// TIA Portal V17 export
// export: Created 2022-03-12T16:05:27.8169496Z, ExportSetting WithDefaults, DisplayName Totally Integrated Automation Portal, DisplayVersion V17, DisplayName TIA Portal Openness, DisplayVersion V17, DisplayName TIA Portal Version Control Interface, DisplayVersion V17, DisplayName STEP 7 Professional, DisplayVersion V17, DisplayName STEP 7 Safety, DisplayVersion V17, DisplayName WinCC Advanced / Unified PC, DisplayVersion V17
FUNCTION_BLOCK "EM01_02_PackML_ModuleSum"   // FB31662, LAD
TITLE = EM01_02_PackML_ModuleSum
{ S7_Optimized_Access := 'TRUE' }
AUTHOR : tech.team.motioncontrol@siemens.com
FAMILY : CPG
VERSION : 1.1
// Support: tech.team.motioncontrol@siemens.com
// stored: AutoNumber true, IsIECCheckEnabled false, IsRetainMemResEnabled false, MemoryReserve 100, SetENOAutomatically false, UDAEnableTagReadback false
   VAR
      statDummyBool { ExternalAccessible := 'False'; ExternalVisible := 'False'; ExternalWritable := 'False'} : Bool;   // dummy bool - placeholder
   END_VAR
BEGIN

REGION Network 1: EM - Reset Command
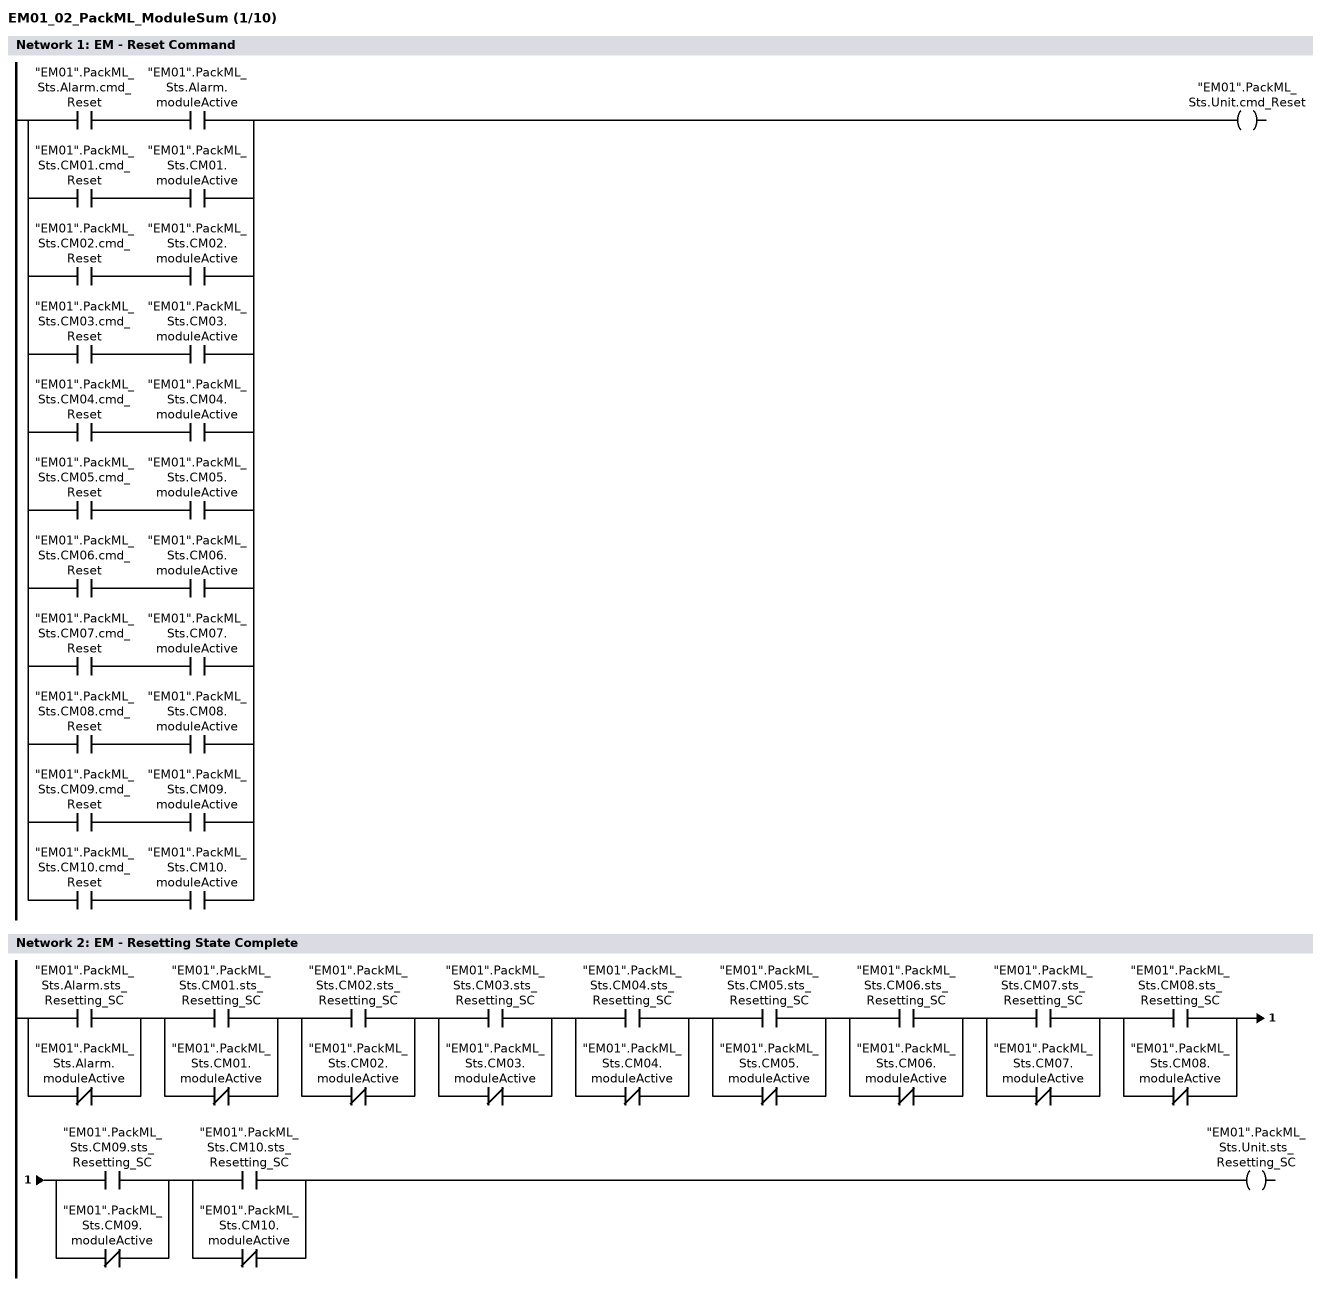
   RUNG wire#powerrail
      Contact( "EM01".PackML_Sts.Alarm.cmd_Reset )
      Contact( "EM01".PackML_Sts.Alarm.moduleActive )
      wire#w1
      Coil( "EM01".PackML_Sts.Unit.cmd_Reset )
   END_RUNG
   RUNG wire#powerrail
      Contact( "EM01".PackML_Sts.CM01.cmd_Reset )
      Contact( "EM01".PackML_Sts.CM01.moduleActive )
   END_RUNG wire#w1
   RUNG wire#powerrail
      Contact( "EM01".PackML_Sts.CM02.cmd_Reset )
      Contact( "EM01".PackML_Sts.CM02.moduleActive )
   END_RUNG wire#w1
   RUNG wire#powerrail
      Contact( "EM01".PackML_Sts.CM03.cmd_Reset )
      Contact( "EM01".PackML_Sts.CM03.moduleActive )
   END_RUNG wire#w1
   RUNG wire#powerrail
      Contact( "EM01".PackML_Sts.CM04.cmd_Reset )
      Contact( "EM01".PackML_Sts.CM04.moduleActive )
   END_RUNG wire#w1
   RUNG wire#powerrail
      Contact( "EM01".PackML_Sts.CM05.cmd_Reset )
      Contact( "EM01".PackML_Sts.CM05.moduleActive )
   END_RUNG wire#w1
   RUNG wire#powerrail
      Contact( "EM01".PackML_Sts.CM06.cmd_Reset )
      Contact( "EM01".PackML_Sts.CM06.moduleActive )
   END_RUNG wire#w1
   RUNG wire#powerrail
      Contact( "EM01".PackML_Sts.CM07.cmd_Reset )
      Contact( "EM01".PackML_Sts.CM07.moduleActive )
   END_RUNG wire#w1
   RUNG wire#powerrail
      Contact( "EM01".PackML_Sts.CM08.cmd_Reset )
      Contact( "EM01".PackML_Sts.CM08.moduleActive )
   END_RUNG wire#w1
   RUNG wire#powerrail
      Contact( "EM01".PackML_Sts.CM09.cmd_Reset )
      Contact( "EM01".PackML_Sts.CM09.moduleActive )
   END_RUNG wire#w1
   RUNG wire#powerrail
      Contact( "EM01".PackML_Sts.CM10.cmd_Reset )
      Contact( "EM01".PackML_Sts.CM10.moduleActive )
   END_RUNG wire#w1
   // the same network as SCL:
   "EM01".PackML_Sts.Unit.cmd_Reset := ("EM01".PackML_Sts.Alarm.cmd_Reset AND "EM01".PackML_Sts.Alarm.moduleActive) OR ("EM01".PackML_Sts.CM01.cmd_Reset AND "EM01".PackML_Sts.CM01.moduleActive) OR ("EM01".PackML_Sts.CM02.cmd_Reset AND "EM01".PackML_Sts.CM02.moduleActive) OR ("EM01".PackML_Sts.CM03.cmd_Reset AND "EM01".PackML_Sts.CM03.moduleActive) OR ("EM01".PackML_Sts.CM04.cmd_Reset AND "EM01".PackML_Sts.CM04.moduleActive) OR ("EM01".PackML_Sts.CM05.cmd_Reset AND "EM01".PackML_Sts.CM05.moduleActive) OR ("EM01".PackML_Sts.CM06.cmd_Reset AND "EM01".PackML_Sts.CM06.moduleActive) OR ("EM01".PackML_Sts.CM07.cmd_Reset AND "EM01".PackML_Sts.CM07.moduleActive) OR ("EM01".PackML_Sts.CM08.cmd_Reset AND "EM01".PackML_Sts.CM08.moduleActive) OR ("EM01".PackML_Sts.CM09.cmd_Reset AND "EM01".PackML_Sts.CM09.moduleActive) OR ("EM01".PackML_Sts.CM10.cmd_Reset AND "EM01".PackML_Sts.CM10.moduleActive);
END_REGION

REGION Network 2: EM - Resetting State Complete
   RUNG wire#powerrail
      Contact( "EM01".PackML_Sts.Alarm.sts_Resetting_SC )
      wire#w1
      Contact( "EM01".PackML_Sts.CM01.sts_Resetting_SC )
      wire#w2
      Contact( "EM01".PackML_Sts.CM02.sts_Resetting_SC )
      wire#w3
      Contact( "EM01".PackML_Sts.CM03.sts_Resetting_SC )
      wire#w4
      Contact( "EM01".PackML_Sts.CM04.sts_Resetting_SC )
      wire#w5
      Contact( "EM01".PackML_Sts.CM05.sts_Resetting_SC )
      wire#w6
      Contact( "EM01".PackML_Sts.CM06.sts_Resetting_SC )
      wire#w7
      Contact( "EM01".PackML_Sts.CM07.sts_Resetting_SC )
      wire#w8
      Contact( "EM01".PackML_Sts.CM08.sts_Resetting_SC )
      wire#w9
      Contact( "EM01".PackML_Sts.CM09.sts_Resetting_SC )
      wire#w10
      Contact( "EM01".PackML_Sts.CM10.sts_Resetting_SC )
      wire#w11
      Coil( "EM01".PackML_Sts.Unit.sts_Resetting_SC )
   END_RUNG
   RUNG wire#powerrail
      I_Contact( "EM01".PackML_Sts.Alarm.moduleActive )
   END_RUNG wire#w1
   RUNG wire#w1
      I_Contact( "EM01".PackML_Sts.CM01.moduleActive )
   END_RUNG wire#w2
   RUNG wire#w2
      I_Contact( "EM01".PackML_Sts.CM02.moduleActive )
   END_RUNG wire#w3
   RUNG wire#w3
      I_Contact( "EM01".PackML_Sts.CM03.moduleActive )
   END_RUNG wire#w4
   RUNG wire#w4
      I_Contact( "EM01".PackML_Sts.CM04.moduleActive )
   END_RUNG wire#w5
   RUNG wire#w5
      I_Contact( "EM01".PackML_Sts.CM05.moduleActive )
   END_RUNG wire#w6
   RUNG wire#w6
      I_Contact( "EM01".PackML_Sts.CM06.moduleActive )
   END_RUNG wire#w7
   RUNG wire#w7
      I_Contact( "EM01".PackML_Sts.CM07.moduleActive )
   END_RUNG wire#w8
   RUNG wire#w8
      I_Contact( "EM01".PackML_Sts.CM08.moduleActive )
   END_RUNG wire#w9
   RUNG wire#w9
      I_Contact( "EM01".PackML_Sts.CM09.moduleActive )
   END_RUNG wire#w10
   RUNG wire#w10
      I_Contact( "EM01".PackML_Sts.CM10.moduleActive )
   END_RUNG wire#w11
   // the same network as SCL:
   "EM01".PackML_Sts.Unit.sts_Resetting_SC := ("EM01".PackML_Sts.Alarm.sts_Resetting_SC OR NOT "EM01".PackML_Sts.Alarm.moduleActive) AND ("EM01".PackML_Sts.CM01.sts_Resetting_SC OR NOT "EM01".PackML_Sts.CM01.moduleActive) AND ("EM01".PackML_Sts.CM02.sts_Resetting_SC OR NOT "EM01".PackML_Sts.CM02.moduleActive) AND ("EM01".PackML_Sts.CM03.sts_Resetting_SC OR NOT "EM01".PackML_Sts.CM03.moduleActive) AND ("EM01".PackML_Sts.CM04.sts_Resetting_SC OR NOT "EM01".PackML_Sts.CM04.moduleActive) AND ("EM01".PackML_Sts.CM05.sts_Resetting_SC OR NOT "EM01".PackML_Sts.CM05.moduleActive) AND ("EM01".PackML_Sts.CM06.sts_Resetting_SC OR NOT "EM01".PackML_Sts.CM06.moduleActive) AND ("EM01".PackML_Sts.CM07.sts_Resetting_SC OR NOT "EM01".PackML_Sts.CM07.moduleActive) AND ("EM01".PackML_Sts.CM08.sts_Resetting_SC OR NOT "EM01".PackML_Sts.CM08.moduleActive) AND ("EM01".PackML_Sts.CM09.sts_Resetting_SC OR NOT "EM01".PackML_Sts.CM09.moduleActive) AND ("EM01".PackML_Sts.CM10.sts_Resetting_SC OR NOT "EM01".PackML_Sts.CM10.moduleActive);
END_REGION

REGION Network 3: EM - Start Command
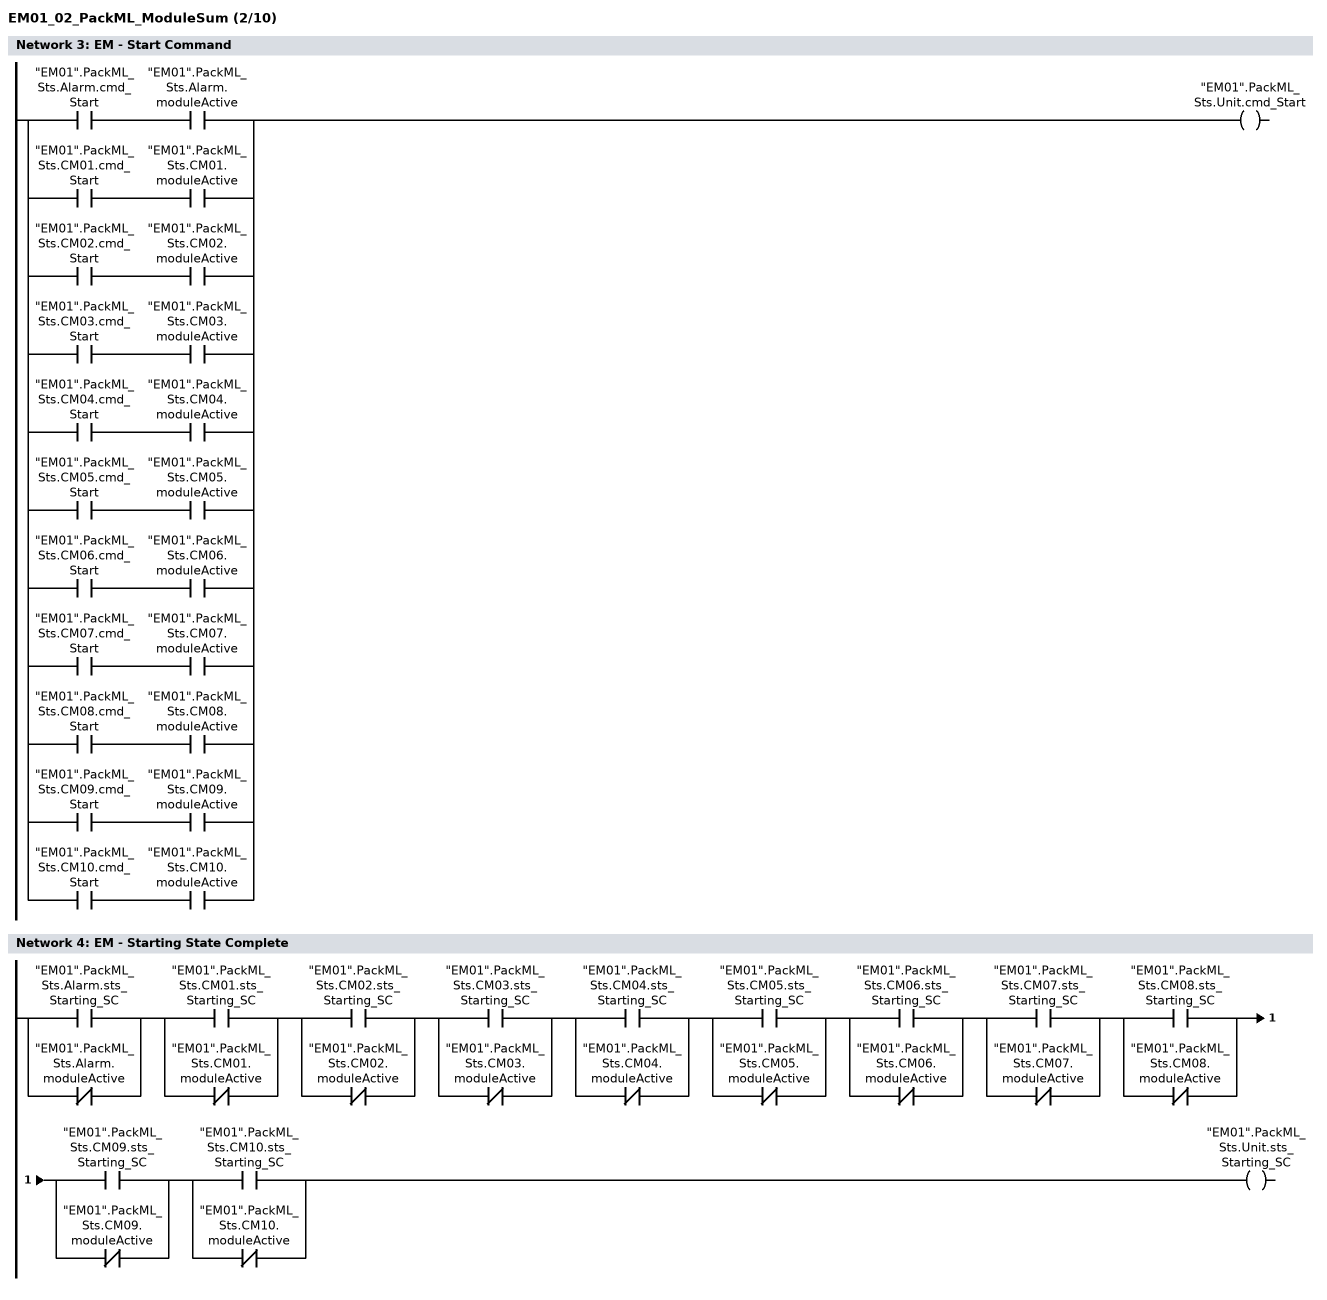
   RUNG wire#powerrail
      Contact( "EM01".PackML_Sts.Alarm.cmd_Start )
      Contact( "EM01".PackML_Sts.Alarm.moduleActive )
      wire#w1
      Coil( "EM01".PackML_Sts.Unit.cmd_Start )
   END_RUNG
   RUNG wire#powerrail
      Contact( "EM01".PackML_Sts.CM01.cmd_Start )
      Contact( "EM01".PackML_Sts.CM01.moduleActive )
   END_RUNG wire#w1
   RUNG wire#powerrail
      Contact( "EM01".PackML_Sts.CM02.cmd_Start )
      Contact( "EM01".PackML_Sts.CM02.moduleActive )
   END_RUNG wire#w1
   RUNG wire#powerrail
      Contact( "EM01".PackML_Sts.CM03.cmd_Start )
      Contact( "EM01".PackML_Sts.CM03.moduleActive )
   END_RUNG wire#w1
   RUNG wire#powerrail
      Contact( "EM01".PackML_Sts.CM04.cmd_Start )
      Contact( "EM01".PackML_Sts.CM04.moduleActive )
   END_RUNG wire#w1
   RUNG wire#powerrail
      Contact( "EM01".PackML_Sts.CM05.cmd_Start )
      Contact( "EM01".PackML_Sts.CM05.moduleActive )
   END_RUNG wire#w1
   RUNG wire#powerrail
      Contact( "EM01".PackML_Sts.CM06.cmd_Start )
      Contact( "EM01".PackML_Sts.CM06.moduleActive )
   END_RUNG wire#w1
   RUNG wire#powerrail
      Contact( "EM01".PackML_Sts.CM07.cmd_Start )
      Contact( "EM01".PackML_Sts.CM07.moduleActive )
   END_RUNG wire#w1
   RUNG wire#powerrail
      Contact( "EM01".PackML_Sts.CM08.cmd_Start )
      Contact( "EM01".PackML_Sts.CM08.moduleActive )
   END_RUNG wire#w1
   RUNG wire#powerrail
      Contact( "EM01".PackML_Sts.CM09.cmd_Start )
      Contact( "EM01".PackML_Sts.CM09.moduleActive )
   END_RUNG wire#w1
   RUNG wire#powerrail
      Contact( "EM01".PackML_Sts.CM10.cmd_Start )
      Contact( "EM01".PackML_Sts.CM10.moduleActive )
   END_RUNG wire#w1
   // the same network as SCL:
   "EM01".PackML_Sts.Unit.cmd_Start := ("EM01".PackML_Sts.Alarm.cmd_Start AND "EM01".PackML_Sts.Alarm.moduleActive) OR ("EM01".PackML_Sts.CM01.cmd_Start AND "EM01".PackML_Sts.CM01.moduleActive) OR ("EM01".PackML_Sts.CM02.cmd_Start AND "EM01".PackML_Sts.CM02.moduleActive) OR ("EM01".PackML_Sts.CM03.cmd_Start AND "EM01".PackML_Sts.CM03.moduleActive) OR ("EM01".PackML_Sts.CM04.cmd_Start AND "EM01".PackML_Sts.CM04.moduleActive) OR ("EM01".PackML_Sts.CM05.cmd_Start AND "EM01".PackML_Sts.CM05.moduleActive) OR ("EM01".PackML_Sts.CM06.cmd_Start AND "EM01".PackML_Sts.CM06.moduleActive) OR ("EM01".PackML_Sts.CM07.cmd_Start AND "EM01".PackML_Sts.CM07.moduleActive) OR ("EM01".PackML_Sts.CM08.cmd_Start AND "EM01".PackML_Sts.CM08.moduleActive) OR ("EM01".PackML_Sts.CM09.cmd_Start AND "EM01".PackML_Sts.CM09.moduleActive) OR ("EM01".PackML_Sts.CM10.cmd_Start AND "EM01".PackML_Sts.CM10.moduleActive);
END_REGION

REGION Network 4: EM - Starting State Complete
   RUNG wire#powerrail
      Contact( "EM01".PackML_Sts.Alarm.sts_Starting_SC )
      wire#w1
      Contact( "EM01".PackML_Sts.CM01.sts_Starting_SC )
      wire#w2
      Contact( "EM01".PackML_Sts.CM02.sts_Starting_SC )
      wire#w3
      Contact( "EM01".PackML_Sts.CM03.sts_Starting_SC )
      wire#w4
      Contact( "EM01".PackML_Sts.CM04.sts_Starting_SC )
      wire#w5
      Contact( "EM01".PackML_Sts.CM05.sts_Starting_SC )
      wire#w6
      Contact( "EM01".PackML_Sts.CM06.sts_Starting_SC )
      wire#w7
      Contact( "EM01".PackML_Sts.CM07.sts_Starting_SC )
      wire#w8
      Contact( "EM01".PackML_Sts.CM08.sts_Starting_SC )
      wire#w9
      Contact( "EM01".PackML_Sts.CM09.sts_Starting_SC )
      wire#w10
      Contact( "EM01".PackML_Sts.CM10.sts_Starting_SC )
      wire#w11
      Coil( "EM01".PackML_Sts.Unit.sts_Starting_SC )
   END_RUNG
   RUNG wire#powerrail
      I_Contact( "EM01".PackML_Sts.Alarm.moduleActive )
   END_RUNG wire#w1
   RUNG wire#w1
      I_Contact( "EM01".PackML_Sts.CM01.moduleActive )
   END_RUNG wire#w2
   RUNG wire#w2
      I_Contact( "EM01".PackML_Sts.CM02.moduleActive )
   END_RUNG wire#w3
   RUNG wire#w3
      I_Contact( "EM01".PackML_Sts.CM03.moduleActive )
   END_RUNG wire#w4
   RUNG wire#w4
      I_Contact( "EM01".PackML_Sts.CM04.moduleActive )
   END_RUNG wire#w5
   RUNG wire#w5
      I_Contact( "EM01".PackML_Sts.CM05.moduleActive )
   END_RUNG wire#w6
   RUNG wire#w6
      I_Contact( "EM01".PackML_Sts.CM06.moduleActive )
   END_RUNG wire#w7
   RUNG wire#w7
      I_Contact( "EM01".PackML_Sts.CM07.moduleActive )
   END_RUNG wire#w8
   RUNG wire#w8
      I_Contact( "EM01".PackML_Sts.CM08.moduleActive )
   END_RUNG wire#w9
   RUNG wire#w9
      I_Contact( "EM01".PackML_Sts.CM09.moduleActive )
   END_RUNG wire#w10
   RUNG wire#w10
      I_Contact( "EM01".PackML_Sts.CM10.moduleActive )
   END_RUNG wire#w11
   // the same network as SCL:
   "EM01".PackML_Sts.Unit.sts_Starting_SC := ("EM01".PackML_Sts.Alarm.sts_Starting_SC OR NOT "EM01".PackML_Sts.Alarm.moduleActive) AND ("EM01".PackML_Sts.CM01.sts_Starting_SC OR NOT "EM01".PackML_Sts.CM01.moduleActive) AND ("EM01".PackML_Sts.CM02.sts_Starting_SC OR NOT "EM01".PackML_Sts.CM02.moduleActive) AND ("EM01".PackML_Sts.CM03.sts_Starting_SC OR NOT "EM01".PackML_Sts.CM03.moduleActive) AND ("EM01".PackML_Sts.CM04.sts_Starting_SC OR NOT "EM01".PackML_Sts.CM04.moduleActive) AND ("EM01".PackML_Sts.CM05.sts_Starting_SC OR NOT "EM01".PackML_Sts.CM05.moduleActive) AND ("EM01".PackML_Sts.CM06.sts_Starting_SC OR NOT "EM01".PackML_Sts.CM06.moduleActive) AND ("EM01".PackML_Sts.CM07.sts_Starting_SC OR NOT "EM01".PackML_Sts.CM07.moduleActive) AND ("EM01".PackML_Sts.CM08.sts_Starting_SC OR NOT "EM01".PackML_Sts.CM08.moduleActive) AND ("EM01".PackML_Sts.CM09.sts_Starting_SC OR NOT "EM01".PackML_Sts.CM09.moduleActive) AND ("EM01".PackML_Sts.CM10.sts_Starting_SC OR NOT "EM01".PackML_Sts.CM10.moduleActive);
END_REGION

REGION Network 5: EM - Stop Command
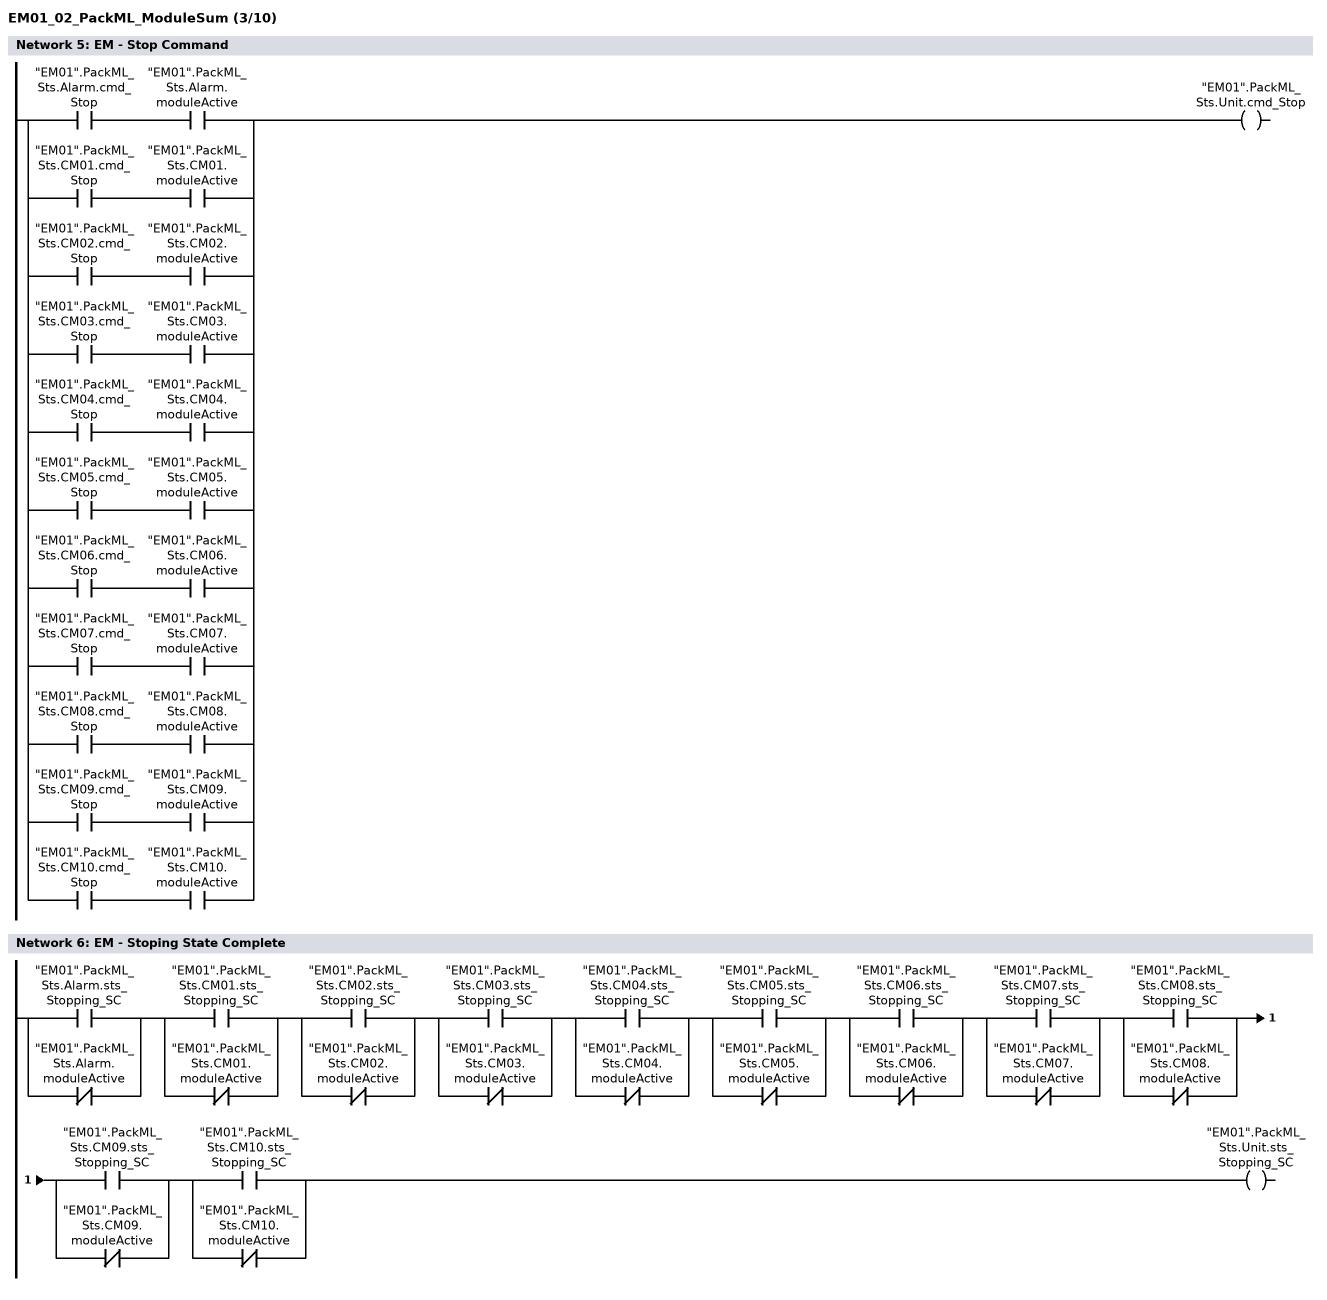
   RUNG wire#powerrail
      Contact( "EM01".PackML_Sts.Alarm.cmd_Stop )
      Contact( "EM01".PackML_Sts.Alarm.moduleActive )
      wire#w1
      Coil( "EM01".PackML_Sts.Unit.cmd_Stop )
   END_RUNG
   RUNG wire#powerrail
      Contact( "EM01".PackML_Sts.CM01.cmd_Stop )
      Contact( "EM01".PackML_Sts.CM01.moduleActive )
   END_RUNG wire#w1
   RUNG wire#powerrail
      Contact( "EM01".PackML_Sts.CM02.cmd_Stop )
      Contact( "EM01".PackML_Sts.CM02.moduleActive )
   END_RUNG wire#w1
   RUNG wire#powerrail
      Contact( "EM01".PackML_Sts.CM03.cmd_Stop )
      Contact( "EM01".PackML_Sts.CM03.moduleActive )
   END_RUNG wire#w1
   RUNG wire#powerrail
      Contact( "EM01".PackML_Sts.CM04.cmd_Stop )
      Contact( "EM01".PackML_Sts.CM04.moduleActive )
   END_RUNG wire#w1
   RUNG wire#powerrail
      Contact( "EM01".PackML_Sts.CM05.cmd_Stop )
      Contact( "EM01".PackML_Sts.CM05.moduleActive )
   END_RUNG wire#w1
   RUNG wire#powerrail
      Contact( "EM01".PackML_Sts.CM06.cmd_Stop )
      Contact( "EM01".PackML_Sts.CM06.moduleActive )
   END_RUNG wire#w1
   RUNG wire#powerrail
      Contact( "EM01".PackML_Sts.CM07.cmd_Stop )
      Contact( "EM01".PackML_Sts.CM07.moduleActive )
   END_RUNG wire#w1
   RUNG wire#powerrail
      Contact( "EM01".PackML_Sts.CM08.cmd_Stop )
      Contact( "EM01".PackML_Sts.CM08.moduleActive )
   END_RUNG wire#w1
   RUNG wire#powerrail
      Contact( "EM01".PackML_Sts.CM09.cmd_Stop )
      Contact( "EM01".PackML_Sts.CM09.moduleActive )
   END_RUNG wire#w1
   RUNG wire#powerrail
      Contact( "EM01".PackML_Sts.CM10.cmd_Stop )
      Contact( "EM01".PackML_Sts.CM10.moduleActive )
   END_RUNG wire#w1
   // the same network as SCL:
   "EM01".PackML_Sts.Unit.cmd_Stop := ("EM01".PackML_Sts.Alarm.cmd_Stop AND "EM01".PackML_Sts.Alarm.moduleActive) OR ("EM01".PackML_Sts.CM01.cmd_Stop AND "EM01".PackML_Sts.CM01.moduleActive) OR ("EM01".PackML_Sts.CM02.cmd_Stop AND "EM01".PackML_Sts.CM02.moduleActive) OR ("EM01".PackML_Sts.CM03.cmd_Stop AND "EM01".PackML_Sts.CM03.moduleActive) OR ("EM01".PackML_Sts.CM04.cmd_Stop AND "EM01".PackML_Sts.CM04.moduleActive) OR ("EM01".PackML_Sts.CM05.cmd_Stop AND "EM01".PackML_Sts.CM05.moduleActive) OR ("EM01".PackML_Sts.CM06.cmd_Stop AND "EM01".PackML_Sts.CM06.moduleActive) OR ("EM01".PackML_Sts.CM07.cmd_Stop AND "EM01".PackML_Sts.CM07.moduleActive) OR ("EM01".PackML_Sts.CM08.cmd_Stop AND "EM01".PackML_Sts.CM08.moduleActive) OR ("EM01".PackML_Sts.CM09.cmd_Stop AND "EM01".PackML_Sts.CM09.moduleActive) OR ("EM01".PackML_Sts.CM10.cmd_Stop AND "EM01".PackML_Sts.CM10.moduleActive);
END_REGION

REGION Network 6: EM - Stoping State Complete
   RUNG wire#powerrail
      Contact( "EM01".PackML_Sts.Alarm.sts_Stopping_SC )
      wire#w1
      Contact( "EM01".PackML_Sts.CM01.sts_Stopping_SC )
      wire#w2
      Contact( "EM01".PackML_Sts.CM02.sts_Stopping_SC )
      wire#w3
      Contact( "EM01".PackML_Sts.CM03.sts_Stopping_SC )
      wire#w4
      Contact( "EM01".PackML_Sts.CM04.sts_Stopping_SC )
      wire#w5
      Contact( "EM01".PackML_Sts.CM05.sts_Stopping_SC )
      wire#w6
      Contact( "EM01".PackML_Sts.CM06.sts_Stopping_SC )
      wire#w7
      Contact( "EM01".PackML_Sts.CM07.sts_Stopping_SC )
      wire#w8
      Contact( "EM01".PackML_Sts.CM08.sts_Stopping_SC )
      wire#w9
      Contact( "EM01".PackML_Sts.CM09.sts_Stopping_SC )
      wire#w10
      Contact( "EM01".PackML_Sts.CM10.sts_Stopping_SC )
      wire#w11
      Coil( "EM01".PackML_Sts.Unit.sts_Stopping_SC )
   END_RUNG
   RUNG wire#powerrail
      I_Contact( "EM01".PackML_Sts.Alarm.moduleActive )
   END_RUNG wire#w1
   RUNG wire#w1
      I_Contact( "EM01".PackML_Sts.CM01.moduleActive )
   END_RUNG wire#w2
   RUNG wire#w2
      I_Contact( "EM01".PackML_Sts.CM02.moduleActive )
   END_RUNG wire#w3
   RUNG wire#w3
      I_Contact( "EM01".PackML_Sts.CM03.moduleActive )
   END_RUNG wire#w4
   RUNG wire#w4
      I_Contact( "EM01".PackML_Sts.CM04.moduleActive )
   END_RUNG wire#w5
   RUNG wire#w5
      I_Contact( "EM01".PackML_Sts.CM05.moduleActive )
   END_RUNG wire#w6
   RUNG wire#w6
      I_Contact( "EM01".PackML_Sts.CM06.moduleActive )
   END_RUNG wire#w7
   RUNG wire#w7
      I_Contact( "EM01".PackML_Sts.CM07.moduleActive )
   END_RUNG wire#w8
   RUNG wire#w8
      I_Contact( "EM01".PackML_Sts.CM08.moduleActive )
   END_RUNG wire#w9
   RUNG wire#w9
      I_Contact( "EM01".PackML_Sts.CM09.moduleActive )
   END_RUNG wire#w10
   RUNG wire#w10
      I_Contact( "EM01".PackML_Sts.CM10.moduleActive )
   END_RUNG wire#w11
   // the same network as SCL:
   "EM01".PackML_Sts.Unit.sts_Stopping_SC := ("EM01".PackML_Sts.Alarm.sts_Stopping_SC OR NOT "EM01".PackML_Sts.Alarm.moduleActive) AND ("EM01".PackML_Sts.CM01.sts_Stopping_SC OR NOT "EM01".PackML_Sts.CM01.moduleActive) AND ("EM01".PackML_Sts.CM02.sts_Stopping_SC OR NOT "EM01".PackML_Sts.CM02.moduleActive) AND ("EM01".PackML_Sts.CM03.sts_Stopping_SC OR NOT "EM01".PackML_Sts.CM03.moduleActive) AND ("EM01".PackML_Sts.CM04.sts_Stopping_SC OR NOT "EM01".PackML_Sts.CM04.moduleActive) AND ("EM01".PackML_Sts.CM05.sts_Stopping_SC OR NOT "EM01".PackML_Sts.CM05.moduleActive) AND ("EM01".PackML_Sts.CM06.sts_Stopping_SC OR NOT "EM01".PackML_Sts.CM06.moduleActive) AND ("EM01".PackML_Sts.CM07.sts_Stopping_SC OR NOT "EM01".PackML_Sts.CM07.moduleActive) AND ("EM01".PackML_Sts.CM08.sts_Stopping_SC OR NOT "EM01".PackML_Sts.CM08.moduleActive) AND ("EM01".PackML_Sts.CM09.sts_Stopping_SC OR NOT "EM01".PackML_Sts.CM09.moduleActive) AND ("EM01".PackML_Sts.CM10.sts_Stopping_SC OR NOT "EM01".PackML_Sts.CM10.moduleActive);
END_REGION

REGION Network 7: EM - Hold Command
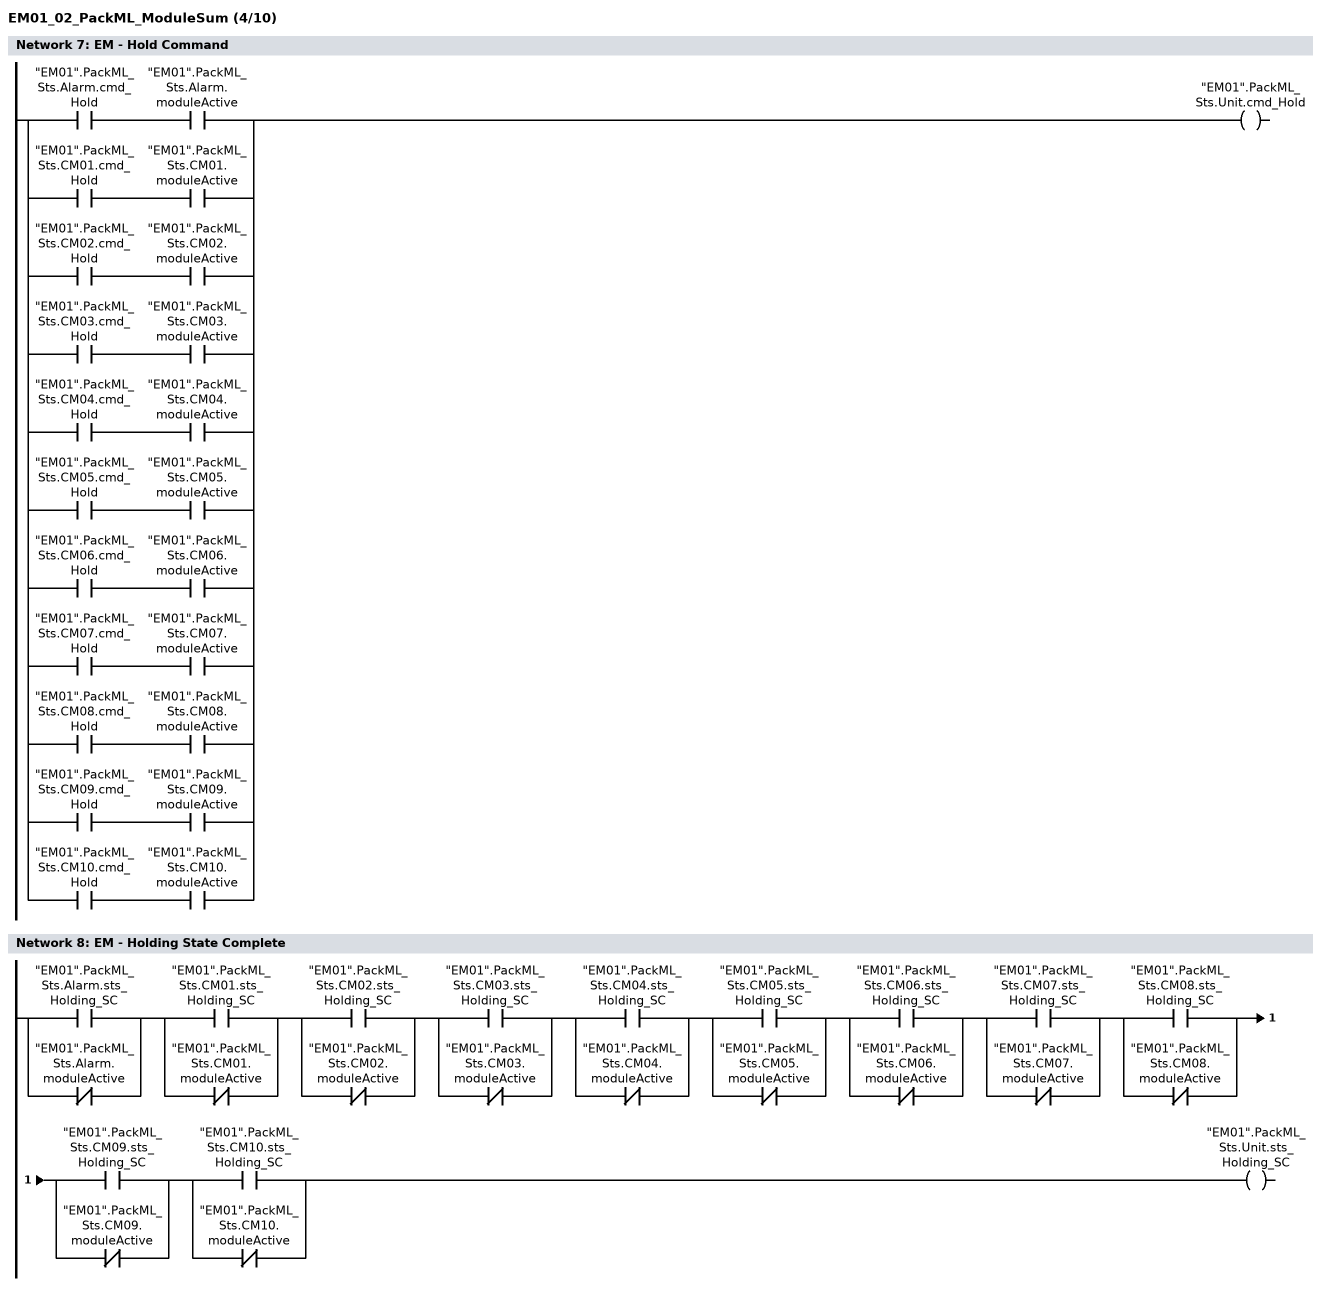
   RUNG wire#powerrail
      Contact( "EM01".PackML_Sts.Alarm.cmd_Hold )
      Contact( "EM01".PackML_Sts.Alarm.moduleActive )
      wire#w1
      Coil( "EM01".PackML_Sts.Unit.cmd_Hold )
   END_RUNG
   RUNG wire#powerrail
      Contact( "EM01".PackML_Sts.CM01.cmd_Hold )
      Contact( "EM01".PackML_Sts.CM01.moduleActive )
   END_RUNG wire#w1
   RUNG wire#powerrail
      Contact( "EM01".PackML_Sts.CM02.cmd_Hold )
      Contact( "EM01".PackML_Sts.CM02.moduleActive )
   END_RUNG wire#w1
   RUNG wire#powerrail
      Contact( "EM01".PackML_Sts.CM03.cmd_Hold )
      Contact( "EM01".PackML_Sts.CM03.moduleActive )
   END_RUNG wire#w1
   RUNG wire#powerrail
      Contact( "EM01".PackML_Sts.CM04.cmd_Hold )
      Contact( "EM01".PackML_Sts.CM04.moduleActive )
   END_RUNG wire#w1
   RUNG wire#powerrail
      Contact( "EM01".PackML_Sts.CM05.cmd_Hold )
      Contact( "EM01".PackML_Sts.CM05.moduleActive )
   END_RUNG wire#w1
   RUNG wire#powerrail
      Contact( "EM01".PackML_Sts.CM06.cmd_Hold )
      Contact( "EM01".PackML_Sts.CM06.moduleActive )
   END_RUNG wire#w1
   RUNG wire#powerrail
      Contact( "EM01".PackML_Sts.CM07.cmd_Hold )
      Contact( "EM01".PackML_Sts.CM07.moduleActive )
   END_RUNG wire#w1
   RUNG wire#powerrail
      Contact( "EM01".PackML_Sts.CM08.cmd_Hold )
      Contact( "EM01".PackML_Sts.CM08.moduleActive )
   END_RUNG wire#w1
   RUNG wire#powerrail
      Contact( "EM01".PackML_Sts.CM09.cmd_Hold )
      Contact( "EM01".PackML_Sts.CM09.moduleActive )
   END_RUNG wire#w1
   RUNG wire#powerrail
      Contact( "EM01".PackML_Sts.CM10.cmd_Hold )
      Contact( "EM01".PackML_Sts.CM10.moduleActive )
   END_RUNG wire#w1
   // the same network as SCL:
   "EM01".PackML_Sts.Unit.cmd_Hold := ("EM01".PackML_Sts.Alarm.cmd_Hold AND "EM01".PackML_Sts.Alarm.moduleActive) OR ("EM01".PackML_Sts.CM01.cmd_Hold AND "EM01".PackML_Sts.CM01.moduleActive) OR ("EM01".PackML_Sts.CM02.cmd_Hold AND "EM01".PackML_Sts.CM02.moduleActive) OR ("EM01".PackML_Sts.CM03.cmd_Hold AND "EM01".PackML_Sts.CM03.moduleActive) OR ("EM01".PackML_Sts.CM04.cmd_Hold AND "EM01".PackML_Sts.CM04.moduleActive) OR ("EM01".PackML_Sts.CM05.cmd_Hold AND "EM01".PackML_Sts.CM05.moduleActive) OR ("EM01".PackML_Sts.CM06.cmd_Hold AND "EM01".PackML_Sts.CM06.moduleActive) OR ("EM01".PackML_Sts.CM07.cmd_Hold AND "EM01".PackML_Sts.CM07.moduleActive) OR ("EM01".PackML_Sts.CM08.cmd_Hold AND "EM01".PackML_Sts.CM08.moduleActive) OR ("EM01".PackML_Sts.CM09.cmd_Hold AND "EM01".PackML_Sts.CM09.moduleActive) OR ("EM01".PackML_Sts.CM10.cmd_Hold AND "EM01".PackML_Sts.CM10.moduleActive);
END_REGION

REGION Network 8: EM - Holding State Complete
   RUNG wire#powerrail
      Contact( "EM01".PackML_Sts.Alarm.sts_Holding_SC )
      wire#w1
      Contact( "EM01".PackML_Sts.CM01.sts_Holding_SC )
      wire#w2
      Contact( "EM01".PackML_Sts.CM02.sts_Holding_SC )
      wire#w3
      Contact( "EM01".PackML_Sts.CM03.sts_Holding_SC )
      wire#w4
      Contact( "EM01".PackML_Sts.CM04.sts_Holding_SC )
      wire#w5
      Contact( "EM01".PackML_Sts.CM05.sts_Holding_SC )
      wire#w6
      Contact( "EM01".PackML_Sts.CM06.sts_Holding_SC )
      wire#w7
      Contact( "EM01".PackML_Sts.CM07.sts_Holding_SC )
      wire#w8
      Contact( "EM01".PackML_Sts.CM08.sts_Holding_SC )
      wire#w9
      Contact( "EM01".PackML_Sts.CM09.sts_Holding_SC )
      wire#w10
      Contact( "EM01".PackML_Sts.CM10.sts_Holding_SC )
      wire#w11
      Coil( "EM01".PackML_Sts.Unit.sts_Holding_SC )
   END_RUNG
   RUNG wire#powerrail
      I_Contact( "EM01".PackML_Sts.Alarm.moduleActive )
   END_RUNG wire#w1
   RUNG wire#w1
      I_Contact( "EM01".PackML_Sts.CM01.moduleActive )
   END_RUNG wire#w2
   RUNG wire#w2
      I_Contact( "EM01".PackML_Sts.CM02.moduleActive )
   END_RUNG wire#w3
   RUNG wire#w3
      I_Contact( "EM01".PackML_Sts.CM03.moduleActive )
   END_RUNG wire#w4
   RUNG wire#w4
      I_Contact( "EM01".PackML_Sts.CM04.moduleActive )
   END_RUNG wire#w5
   RUNG wire#w5
      I_Contact( "EM01".PackML_Sts.CM05.moduleActive )
   END_RUNG wire#w6
   RUNG wire#w6
      I_Contact( "EM01".PackML_Sts.CM06.moduleActive )
   END_RUNG wire#w7
   RUNG wire#w7
      I_Contact( "EM01".PackML_Sts.CM07.moduleActive )
   END_RUNG wire#w8
   RUNG wire#w8
      I_Contact( "EM01".PackML_Sts.CM08.moduleActive )
   END_RUNG wire#w9
   RUNG wire#w9
      I_Contact( "EM01".PackML_Sts.CM09.moduleActive )
   END_RUNG wire#w10
   RUNG wire#w10
      I_Contact( "EM01".PackML_Sts.CM10.moduleActive )
   END_RUNG wire#w11
   // the same network as SCL:
   "EM01".PackML_Sts.Unit.sts_Holding_SC := ("EM01".PackML_Sts.Alarm.sts_Holding_SC OR NOT "EM01".PackML_Sts.Alarm.moduleActive) AND ("EM01".PackML_Sts.CM01.sts_Holding_SC OR NOT "EM01".PackML_Sts.CM01.moduleActive) AND ("EM01".PackML_Sts.CM02.sts_Holding_SC OR NOT "EM01".PackML_Sts.CM02.moduleActive) AND ("EM01".PackML_Sts.CM03.sts_Holding_SC OR NOT "EM01".PackML_Sts.CM03.moduleActive) AND ("EM01".PackML_Sts.CM04.sts_Holding_SC OR NOT "EM01".PackML_Sts.CM04.moduleActive) AND ("EM01".PackML_Sts.CM05.sts_Holding_SC OR NOT "EM01".PackML_Sts.CM05.moduleActive) AND ("EM01".PackML_Sts.CM06.sts_Holding_SC OR NOT "EM01".PackML_Sts.CM06.moduleActive) AND ("EM01".PackML_Sts.CM07.sts_Holding_SC OR NOT "EM01".PackML_Sts.CM07.moduleActive) AND ("EM01".PackML_Sts.CM08.sts_Holding_SC OR NOT "EM01".PackML_Sts.CM08.moduleActive) AND ("EM01".PackML_Sts.CM09.sts_Holding_SC OR NOT "EM01".PackML_Sts.CM09.moduleActive) AND ("EM01".PackML_Sts.CM10.sts_Holding_SC OR NOT "EM01".PackML_Sts.CM10.moduleActive);
END_REGION

REGION Network 9: EM - UnHold Command
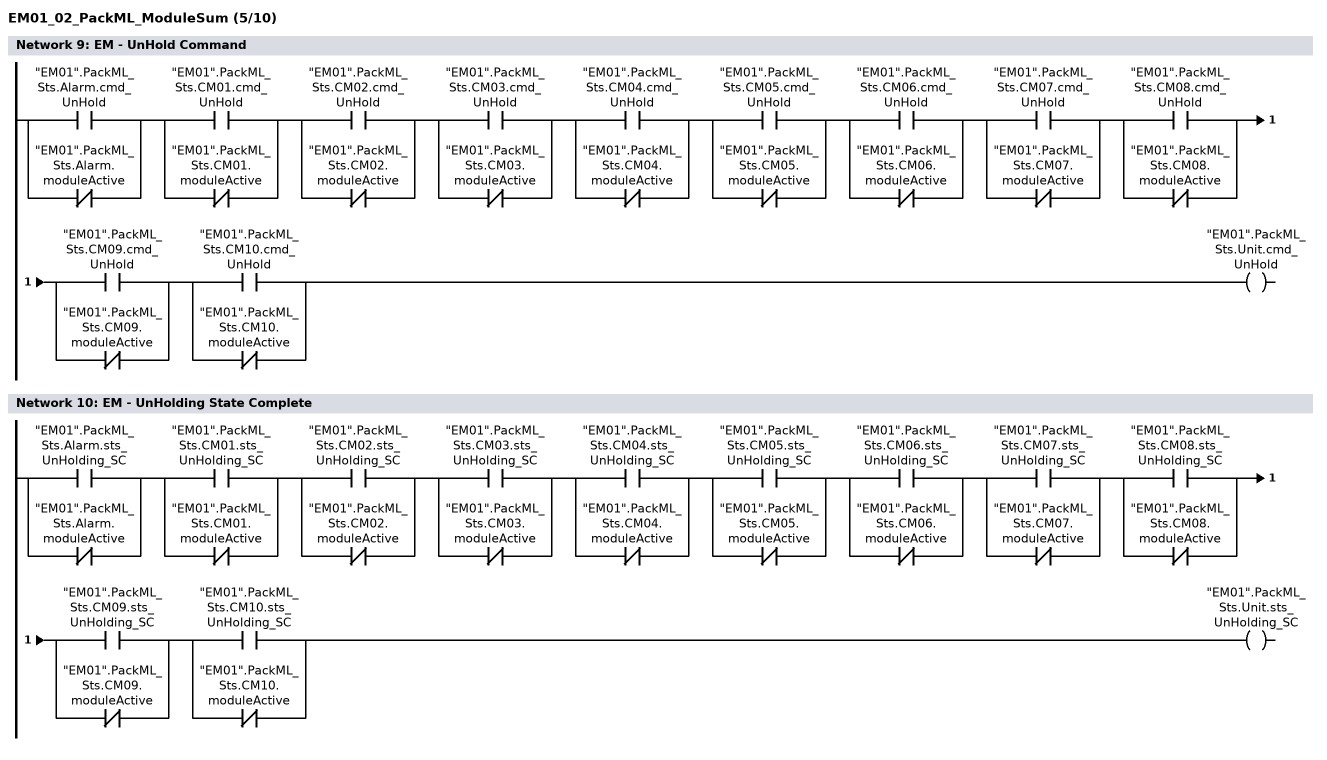
   RUNG wire#powerrail
      Contact( "EM01".PackML_Sts.Alarm.cmd_UnHold )
      wire#w1
      Contact( "EM01".PackML_Sts.CM01.cmd_UnHold )
      wire#w2
      Contact( "EM01".PackML_Sts.CM02.cmd_UnHold )
      wire#w3
      Contact( "EM01".PackML_Sts.CM03.cmd_UnHold )
      wire#w4
      Contact( "EM01".PackML_Sts.CM04.cmd_UnHold )
      wire#w5
      Contact( "EM01".PackML_Sts.CM05.cmd_UnHold )
      wire#w6
      Contact( "EM01".PackML_Sts.CM06.cmd_UnHold )
      wire#w7
      Contact( "EM01".PackML_Sts.CM07.cmd_UnHold )
      wire#w8
      Contact( "EM01".PackML_Sts.CM08.cmd_UnHold )
      wire#w9
      Contact( "EM01".PackML_Sts.CM09.cmd_UnHold )
      wire#w10
      Contact( "EM01".PackML_Sts.CM10.cmd_UnHold )
      wire#w11
      Coil( "EM01".PackML_Sts.Unit.cmd_UnHold )
   END_RUNG
   RUNG wire#powerrail
      I_Contact( "EM01".PackML_Sts.Alarm.moduleActive )
   END_RUNG wire#w1
   RUNG wire#w1
      I_Contact( "EM01".PackML_Sts.CM01.moduleActive )
   END_RUNG wire#w2
   RUNG wire#w2
      I_Contact( "EM01".PackML_Sts.CM02.moduleActive )
   END_RUNG wire#w3
   RUNG wire#w3
      I_Contact( "EM01".PackML_Sts.CM03.moduleActive )
   END_RUNG wire#w4
   RUNG wire#w4
      I_Contact( "EM01".PackML_Sts.CM04.moduleActive )
   END_RUNG wire#w5
   RUNG wire#w5
      I_Contact( "EM01".PackML_Sts.CM05.moduleActive )
   END_RUNG wire#w6
   RUNG wire#w6
      I_Contact( "EM01".PackML_Sts.CM06.moduleActive )
   END_RUNG wire#w7
   RUNG wire#w7
      I_Contact( "EM01".PackML_Sts.CM07.moduleActive )
   END_RUNG wire#w8
   RUNG wire#w8
      I_Contact( "EM01".PackML_Sts.CM08.moduleActive )
   END_RUNG wire#w9
   RUNG wire#w9
      I_Contact( "EM01".PackML_Sts.CM09.moduleActive )
   END_RUNG wire#w10
   RUNG wire#w10
      I_Contact( "EM01".PackML_Sts.CM10.moduleActive )
   END_RUNG wire#w11
   // the same network as SCL:
   "EM01".PackML_Sts.Unit.cmd_UnHold := ("EM01".PackML_Sts.Alarm.cmd_UnHold OR NOT "EM01".PackML_Sts.Alarm.moduleActive) AND ("EM01".PackML_Sts.CM01.cmd_UnHold OR NOT "EM01".PackML_Sts.CM01.moduleActive) AND ("EM01".PackML_Sts.CM02.cmd_UnHold OR NOT "EM01".PackML_Sts.CM02.moduleActive) AND ("EM01".PackML_Sts.CM03.cmd_UnHold OR NOT "EM01".PackML_Sts.CM03.moduleActive) AND ("EM01".PackML_Sts.CM04.cmd_UnHold OR NOT "EM01".PackML_Sts.CM04.moduleActive) AND ("EM01".PackML_Sts.CM05.cmd_UnHold OR NOT "EM01".PackML_Sts.CM05.moduleActive) AND ("EM01".PackML_Sts.CM06.cmd_UnHold OR NOT "EM01".PackML_Sts.CM06.moduleActive) AND ("EM01".PackML_Sts.CM07.cmd_UnHold OR NOT "EM01".PackML_Sts.CM07.moduleActive) AND ("EM01".PackML_Sts.CM08.cmd_UnHold OR NOT "EM01".PackML_Sts.CM08.moduleActive) AND ("EM01".PackML_Sts.CM09.cmd_UnHold OR NOT "EM01".PackML_Sts.CM09.moduleActive) AND ("EM01".PackML_Sts.CM10.cmd_UnHold OR NOT "EM01".PackML_Sts.CM10.moduleActive);
END_REGION

REGION Network 10: EM - UnHolding State Complete
   RUNG wire#powerrail
      Contact( "EM01".PackML_Sts.Alarm.sts_UnHolding_SC )
      wire#w1
      Contact( "EM01".PackML_Sts.CM01.sts_UnHolding_SC )
      wire#w2
      Contact( "EM01".PackML_Sts.CM02.sts_UnHolding_SC )
      wire#w3
      Contact( "EM01".PackML_Sts.CM03.sts_UnHolding_SC )
      wire#w4
      Contact( "EM01".PackML_Sts.CM04.sts_UnHolding_SC )
      wire#w5
      Contact( "EM01".PackML_Sts.CM05.sts_UnHolding_SC )
      wire#w6
      Contact( "EM01".PackML_Sts.CM06.sts_UnHolding_SC )
      wire#w7
      Contact( "EM01".PackML_Sts.CM07.sts_UnHolding_SC )
      wire#w8
      Contact( "EM01".PackML_Sts.CM08.sts_UnHolding_SC )
      wire#w9
      Contact( "EM01".PackML_Sts.CM09.sts_UnHolding_SC )
      wire#w10
      Contact( "EM01".PackML_Sts.CM10.sts_UnHolding_SC )
      wire#w11
      Coil( "EM01".PackML_Sts.Unit.sts_UnHolding_SC )
   END_RUNG
   RUNG wire#powerrail
      I_Contact( "EM01".PackML_Sts.Alarm.moduleActive )
   END_RUNG wire#w1
   RUNG wire#w1
      I_Contact( "EM01".PackML_Sts.CM01.moduleActive )
   END_RUNG wire#w2
   RUNG wire#w2
      I_Contact( "EM01".PackML_Sts.CM02.moduleActive )
   END_RUNG wire#w3
   RUNG wire#w3
      I_Contact( "EM01".PackML_Sts.CM03.moduleActive )
   END_RUNG wire#w4
   RUNG wire#w4
      I_Contact( "EM01".PackML_Sts.CM04.moduleActive )
   END_RUNG wire#w5
   RUNG wire#w5
      I_Contact( "EM01".PackML_Sts.CM05.moduleActive )
   END_RUNG wire#w6
   RUNG wire#w6
      I_Contact( "EM01".PackML_Sts.CM06.moduleActive )
   END_RUNG wire#w7
   RUNG wire#w7
      I_Contact( "EM01".PackML_Sts.CM07.moduleActive )
   END_RUNG wire#w8
   RUNG wire#w8
      I_Contact( "EM01".PackML_Sts.CM08.moduleActive )
   END_RUNG wire#w9
   RUNG wire#w9
      I_Contact( "EM01".PackML_Sts.CM09.moduleActive )
   END_RUNG wire#w10
   RUNG wire#w10
      I_Contact( "EM01".PackML_Sts.CM10.moduleActive )
   END_RUNG wire#w11
   // the same network as SCL:
   "EM01".PackML_Sts.Unit.sts_UnHolding_SC := ("EM01".PackML_Sts.Alarm.sts_UnHolding_SC OR NOT "EM01".PackML_Sts.Alarm.moduleActive) AND ("EM01".PackML_Sts.CM01.sts_UnHolding_SC OR NOT "EM01".PackML_Sts.CM01.moduleActive) AND ("EM01".PackML_Sts.CM02.sts_UnHolding_SC OR NOT "EM01".PackML_Sts.CM02.moduleActive) AND ("EM01".PackML_Sts.CM03.sts_UnHolding_SC OR NOT "EM01".PackML_Sts.CM03.moduleActive) AND ("EM01".PackML_Sts.CM04.sts_UnHolding_SC OR NOT "EM01".PackML_Sts.CM04.moduleActive) AND ("EM01".PackML_Sts.CM05.sts_UnHolding_SC OR NOT "EM01".PackML_Sts.CM05.moduleActive) AND ("EM01".PackML_Sts.CM06.sts_UnHolding_SC OR NOT "EM01".PackML_Sts.CM06.moduleActive) AND ("EM01".PackML_Sts.CM07.sts_UnHolding_SC OR NOT "EM01".PackML_Sts.CM07.moduleActive) AND ("EM01".PackML_Sts.CM08.sts_UnHolding_SC OR NOT "EM01".PackML_Sts.CM08.moduleActive) AND ("EM01".PackML_Sts.CM09.sts_UnHolding_SC OR NOT "EM01".PackML_Sts.CM09.moduleActive) AND ("EM01".PackML_Sts.CM10.sts_UnHolding_SC OR NOT "EM01".PackML_Sts.CM10.moduleActive);
END_REGION

REGION Network 11: EM - Suspend Command
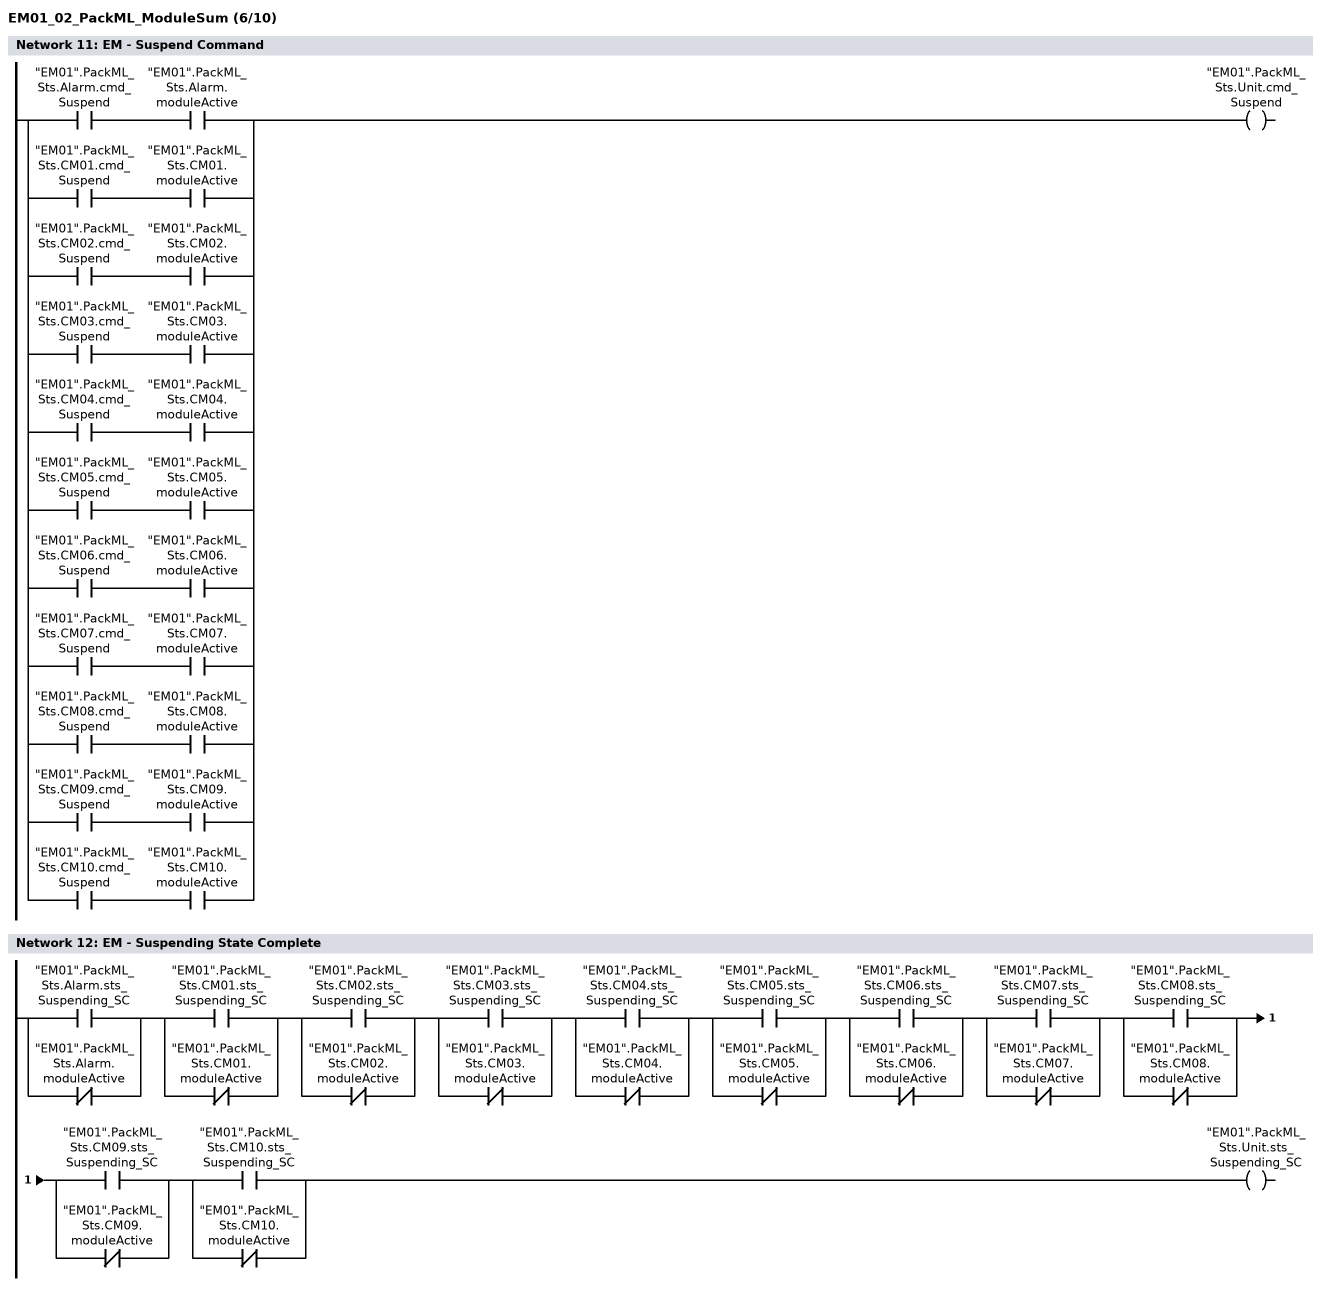
   RUNG wire#powerrail
      Contact( "EM01".PackML_Sts.Alarm.cmd_Suspend )
      Contact( "EM01".PackML_Sts.Alarm.moduleActive )
      wire#w1
      Coil( "EM01".PackML_Sts.Unit.cmd_Suspend )
   END_RUNG
   RUNG wire#powerrail
      Contact( "EM01".PackML_Sts.CM01.cmd_Suspend )
      Contact( "EM01".PackML_Sts.CM01.moduleActive )
   END_RUNG wire#w1
   RUNG wire#powerrail
      Contact( "EM01".PackML_Sts.CM02.cmd_Suspend )
      Contact( "EM01".PackML_Sts.CM02.moduleActive )
   END_RUNG wire#w1
   RUNG wire#powerrail
      Contact( "EM01".PackML_Sts.CM03.cmd_Suspend )
      Contact( "EM01".PackML_Sts.CM03.moduleActive )
   END_RUNG wire#w1
   RUNG wire#powerrail
      Contact( "EM01".PackML_Sts.CM04.cmd_Suspend )
      Contact( "EM01".PackML_Sts.CM04.moduleActive )
   END_RUNG wire#w1
   RUNG wire#powerrail
      Contact( "EM01".PackML_Sts.CM05.cmd_Suspend )
      Contact( "EM01".PackML_Sts.CM05.moduleActive )
   END_RUNG wire#w1
   RUNG wire#powerrail
      Contact( "EM01".PackML_Sts.CM06.cmd_Suspend )
      Contact( "EM01".PackML_Sts.CM06.moduleActive )
   END_RUNG wire#w1
   RUNG wire#powerrail
      Contact( "EM01".PackML_Sts.CM07.cmd_Suspend )
      Contact( "EM01".PackML_Sts.CM07.moduleActive )
   END_RUNG wire#w1
   RUNG wire#powerrail
      Contact( "EM01".PackML_Sts.CM08.cmd_Suspend )
      Contact( "EM01".PackML_Sts.CM08.moduleActive )
   END_RUNG wire#w1
   RUNG wire#powerrail
      Contact( "EM01".PackML_Sts.CM09.cmd_Suspend )
      Contact( "EM01".PackML_Sts.CM09.moduleActive )
   END_RUNG wire#w1
   RUNG wire#powerrail
      Contact( "EM01".PackML_Sts.CM10.cmd_Suspend )
      Contact( "EM01".PackML_Sts.CM10.moduleActive )
   END_RUNG wire#w1
   // the same network as SCL:
   "EM01".PackML_Sts.Unit.cmd_Suspend := ("EM01".PackML_Sts.Alarm.cmd_Suspend AND "EM01".PackML_Sts.Alarm.moduleActive) OR ("EM01".PackML_Sts.CM01.cmd_Suspend AND "EM01".PackML_Sts.CM01.moduleActive) OR ("EM01".PackML_Sts.CM02.cmd_Suspend AND "EM01".PackML_Sts.CM02.moduleActive) OR ("EM01".PackML_Sts.CM03.cmd_Suspend AND "EM01".PackML_Sts.CM03.moduleActive) OR ("EM01".PackML_Sts.CM04.cmd_Suspend AND "EM01".PackML_Sts.CM04.moduleActive) OR ("EM01".PackML_Sts.CM05.cmd_Suspend AND "EM01".PackML_Sts.CM05.moduleActive) OR ("EM01".PackML_Sts.CM06.cmd_Suspend AND "EM01".PackML_Sts.CM06.moduleActive) OR ("EM01".PackML_Sts.CM07.cmd_Suspend AND "EM01".PackML_Sts.CM07.moduleActive) OR ("EM01".PackML_Sts.CM08.cmd_Suspend AND "EM01".PackML_Sts.CM08.moduleActive) OR ("EM01".PackML_Sts.CM09.cmd_Suspend AND "EM01".PackML_Sts.CM09.moduleActive) OR ("EM01".PackML_Sts.CM10.cmd_Suspend AND "EM01".PackML_Sts.CM10.moduleActive);
END_REGION

REGION Network 12: EM - Suspending State Complete
   RUNG wire#powerrail
      Contact( "EM01".PackML_Sts.Alarm.sts_Suspending_SC )
      wire#w1
      Contact( "EM01".PackML_Sts.CM01.sts_Suspending_SC )
      wire#w2
      Contact( "EM01".PackML_Sts.CM02.sts_Suspending_SC )
      wire#w3
      Contact( "EM01".PackML_Sts.CM03.sts_Suspending_SC )
      wire#w4
      Contact( "EM01".PackML_Sts.CM04.sts_Suspending_SC )
      wire#w5
      Contact( "EM01".PackML_Sts.CM05.sts_Suspending_SC )
      wire#w6
      Contact( "EM01".PackML_Sts.CM06.sts_Suspending_SC )
      wire#w7
      Contact( "EM01".PackML_Sts.CM07.sts_Suspending_SC )
      wire#w8
      Contact( "EM01".PackML_Sts.CM08.sts_Suspending_SC )
      wire#w9
      Contact( "EM01".PackML_Sts.CM09.sts_Suspending_SC )
      wire#w10
      Contact( "EM01".PackML_Sts.CM10.sts_Suspending_SC )
      wire#w11
      Coil( "EM01".PackML_Sts.Unit.sts_Suspending_SC )
   END_RUNG
   RUNG wire#powerrail
      I_Contact( "EM01".PackML_Sts.Alarm.moduleActive )
   END_RUNG wire#w1
   RUNG wire#w1
      I_Contact( "EM01".PackML_Sts.CM01.moduleActive )
   END_RUNG wire#w2
   RUNG wire#w2
      I_Contact( "EM01".PackML_Sts.CM02.moduleActive )
   END_RUNG wire#w3
   RUNG wire#w3
      I_Contact( "EM01".PackML_Sts.CM03.moduleActive )
   END_RUNG wire#w4
   RUNG wire#w4
      I_Contact( "EM01".PackML_Sts.CM04.moduleActive )
   END_RUNG wire#w5
   RUNG wire#w5
      I_Contact( "EM01".PackML_Sts.CM05.moduleActive )
   END_RUNG wire#w6
   RUNG wire#w6
      I_Contact( "EM01".PackML_Sts.CM06.moduleActive )
   END_RUNG wire#w7
   RUNG wire#w7
      I_Contact( "EM01".PackML_Sts.CM07.moduleActive )
   END_RUNG wire#w8
   RUNG wire#w8
      I_Contact( "EM01".PackML_Sts.CM08.moduleActive )
   END_RUNG wire#w9
   RUNG wire#w9
      I_Contact( "EM01".PackML_Sts.CM09.moduleActive )
   END_RUNG wire#w10
   RUNG wire#w10
      I_Contact( "EM01".PackML_Sts.CM10.moduleActive )
   END_RUNG wire#w11
   // the same network as SCL:
   "EM01".PackML_Sts.Unit.sts_Suspending_SC := ("EM01".PackML_Sts.Alarm.sts_Suspending_SC OR NOT "EM01".PackML_Sts.Alarm.moduleActive) AND ("EM01".PackML_Sts.CM01.sts_Suspending_SC OR NOT "EM01".PackML_Sts.CM01.moduleActive) AND ("EM01".PackML_Sts.CM02.sts_Suspending_SC OR NOT "EM01".PackML_Sts.CM02.moduleActive) AND ("EM01".PackML_Sts.CM03.sts_Suspending_SC OR NOT "EM01".PackML_Sts.CM03.moduleActive) AND ("EM01".PackML_Sts.CM04.sts_Suspending_SC OR NOT "EM01".PackML_Sts.CM04.moduleActive) AND ("EM01".PackML_Sts.CM05.sts_Suspending_SC OR NOT "EM01".PackML_Sts.CM05.moduleActive) AND ("EM01".PackML_Sts.CM06.sts_Suspending_SC OR NOT "EM01".PackML_Sts.CM06.moduleActive) AND ("EM01".PackML_Sts.CM07.sts_Suspending_SC OR NOT "EM01".PackML_Sts.CM07.moduleActive) AND ("EM01".PackML_Sts.CM08.sts_Suspending_SC OR NOT "EM01".PackML_Sts.CM08.moduleActive) AND ("EM01".PackML_Sts.CM09.sts_Suspending_SC OR NOT "EM01".PackML_Sts.CM09.moduleActive) AND ("EM01".PackML_Sts.CM10.sts_Suspending_SC OR NOT "EM01".PackML_Sts.CM10.moduleActive);
END_REGION

REGION Network 13: EM - UnSuspend Command
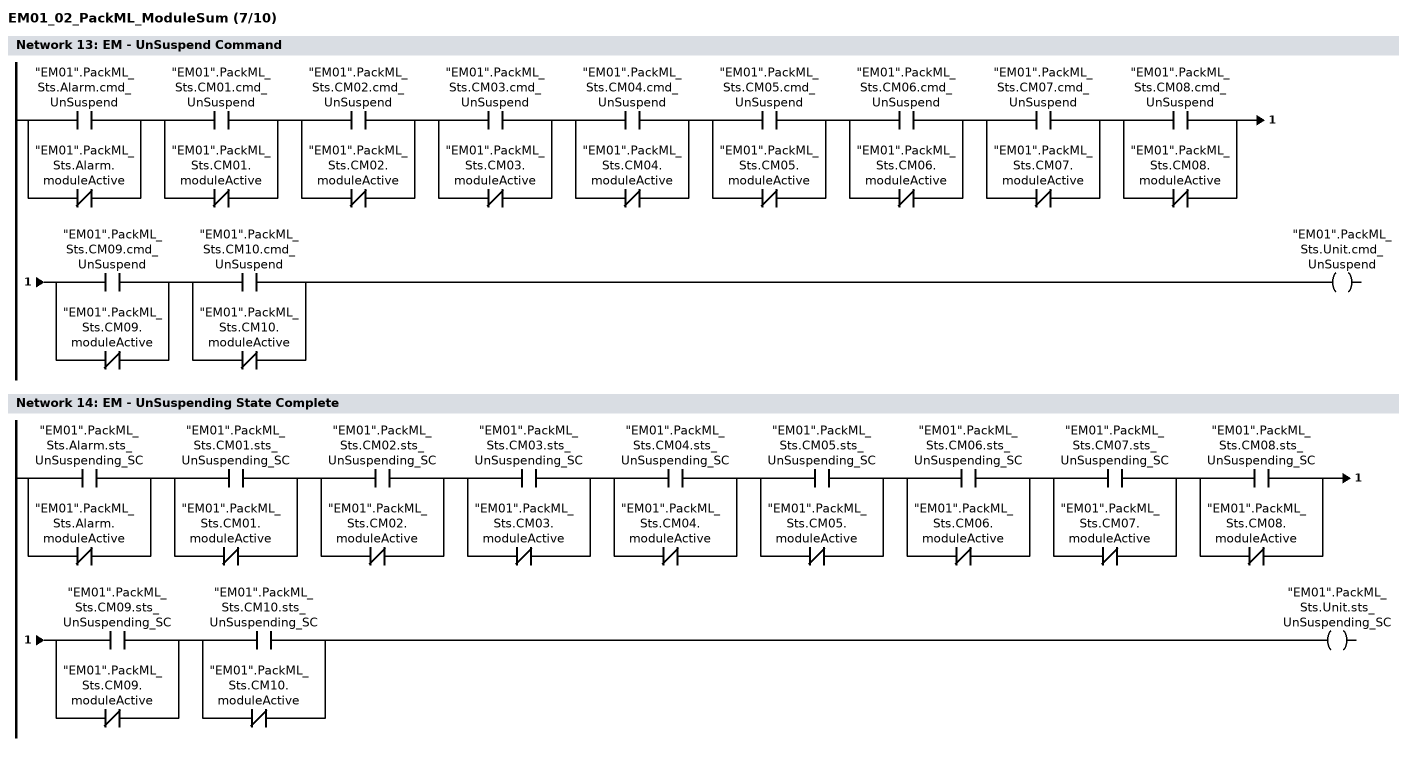
   RUNG wire#powerrail
      Contact( "EM01".PackML_Sts.Alarm.cmd_UnSuspend )
      wire#w1
      Contact( "EM01".PackML_Sts.CM01.cmd_UnSuspend )
      wire#w2
      Contact( "EM01".PackML_Sts.CM02.cmd_UnSuspend )
      wire#w3
      Contact( "EM01".PackML_Sts.CM03.cmd_UnSuspend )
      wire#w4
      Contact( "EM01".PackML_Sts.CM04.cmd_UnSuspend )
      wire#w5
      Contact( "EM01".PackML_Sts.CM05.cmd_UnSuspend )
      wire#w6
      Contact( "EM01".PackML_Sts.CM06.cmd_UnSuspend )
      wire#w7
      Contact( "EM01".PackML_Sts.CM07.cmd_UnSuspend )
      wire#w8
      Contact( "EM01".PackML_Sts.CM08.cmd_UnSuspend )
      wire#w9
      Contact( "EM01".PackML_Sts.CM09.cmd_UnSuspend )
      wire#w10
      Contact( "EM01".PackML_Sts.CM10.cmd_UnSuspend )
      wire#w11
      Coil( "EM01".PackML_Sts.Unit.cmd_UnSuspend )
   END_RUNG
   RUNG wire#powerrail
      I_Contact( "EM01".PackML_Sts.Alarm.moduleActive )
   END_RUNG wire#w1
   RUNG wire#w1
      I_Contact( "EM01".PackML_Sts.CM01.moduleActive )
   END_RUNG wire#w2
   RUNG wire#w2
      I_Contact( "EM01".PackML_Sts.CM02.moduleActive )
   END_RUNG wire#w3
   RUNG wire#w3
      I_Contact( "EM01".PackML_Sts.CM03.moduleActive )
   END_RUNG wire#w4
   RUNG wire#w4
      I_Contact( "EM01".PackML_Sts.CM04.moduleActive )
   END_RUNG wire#w5
   RUNG wire#w5
      I_Contact( "EM01".PackML_Sts.CM05.moduleActive )
   END_RUNG wire#w6
   RUNG wire#w6
      I_Contact( "EM01".PackML_Sts.CM06.moduleActive )
   END_RUNG wire#w7
   RUNG wire#w7
      I_Contact( "EM01".PackML_Sts.CM07.moduleActive )
   END_RUNG wire#w8
   RUNG wire#w8
      I_Contact( "EM01".PackML_Sts.CM08.moduleActive )
   END_RUNG wire#w9
   RUNG wire#w9
      I_Contact( "EM01".PackML_Sts.CM09.moduleActive )
   END_RUNG wire#w10
   RUNG wire#w10
      I_Contact( "EM01".PackML_Sts.CM10.moduleActive )
   END_RUNG wire#w11
   // the same network as SCL:
   "EM01".PackML_Sts.Unit.cmd_UnSuspend := ("EM01".PackML_Sts.Alarm.cmd_UnSuspend OR NOT "EM01".PackML_Sts.Alarm.moduleActive) AND ("EM01".PackML_Sts.CM01.cmd_UnSuspend OR NOT "EM01".PackML_Sts.CM01.moduleActive) AND ("EM01".PackML_Sts.CM02.cmd_UnSuspend OR NOT "EM01".PackML_Sts.CM02.moduleActive) AND ("EM01".PackML_Sts.CM03.cmd_UnSuspend OR NOT "EM01".PackML_Sts.CM03.moduleActive) AND ("EM01".PackML_Sts.CM04.cmd_UnSuspend OR NOT "EM01".PackML_Sts.CM04.moduleActive) AND ("EM01".PackML_Sts.CM05.cmd_UnSuspend OR NOT "EM01".PackML_Sts.CM05.moduleActive) AND ("EM01".PackML_Sts.CM06.cmd_UnSuspend OR NOT "EM01".PackML_Sts.CM06.moduleActive) AND ("EM01".PackML_Sts.CM07.cmd_UnSuspend OR NOT "EM01".PackML_Sts.CM07.moduleActive) AND ("EM01".PackML_Sts.CM08.cmd_UnSuspend OR NOT "EM01".PackML_Sts.CM08.moduleActive) AND ("EM01".PackML_Sts.CM09.cmd_UnSuspend OR NOT "EM01".PackML_Sts.CM09.moduleActive) AND ("EM01".PackML_Sts.CM10.cmd_UnSuspend OR NOT "EM01".PackML_Sts.CM10.moduleActive);
END_REGION

REGION Network 14: EM - UnSuspending State Complete
   RUNG wire#powerrail
      Contact( "EM01".PackML_Sts.Alarm.sts_UnSuspending_SC )
      wire#w1
      Contact( "EM01".PackML_Sts.CM01.sts_UnSuspending_SC )
      wire#w2
      Contact( "EM01".PackML_Sts.CM02.sts_UnSuspending_SC )
      wire#w3
      Contact( "EM01".PackML_Sts.CM03.sts_UnSuspending_SC )
      wire#w4
      Contact( "EM01".PackML_Sts.CM04.sts_UnSuspending_SC )
      wire#w5
      Contact( "EM01".PackML_Sts.CM05.sts_UnSuspending_SC )
      wire#w6
      Contact( "EM01".PackML_Sts.CM06.sts_UnSuspending_SC )
      wire#w7
      Contact( "EM01".PackML_Sts.CM07.sts_UnSuspending_SC )
      wire#w8
      Contact( "EM01".PackML_Sts.CM08.sts_UnSuspending_SC )
      wire#w9
      Contact( "EM01".PackML_Sts.CM09.sts_UnSuspending_SC )
      wire#w10
      Contact( "EM01".PackML_Sts.CM10.sts_UnSuspending_SC )
      wire#w11
      Coil( "EM01".PackML_Sts.Unit.sts_UnSuspending_SC )
   END_RUNG
   RUNG wire#powerrail
      I_Contact( "EM01".PackML_Sts.Alarm.moduleActive )
   END_RUNG wire#w1
   RUNG wire#w1
      I_Contact( "EM01".PackML_Sts.CM01.moduleActive )
   END_RUNG wire#w2
   RUNG wire#w2
      I_Contact( "EM01".PackML_Sts.CM02.moduleActive )
   END_RUNG wire#w3
   RUNG wire#w3
      I_Contact( "EM01".PackML_Sts.CM03.moduleActive )
   END_RUNG wire#w4
   RUNG wire#w4
      I_Contact( "EM01".PackML_Sts.CM04.moduleActive )
   END_RUNG wire#w5
   RUNG wire#w5
      I_Contact( "EM01".PackML_Sts.CM05.moduleActive )
   END_RUNG wire#w6
   RUNG wire#w6
      I_Contact( "EM01".PackML_Sts.CM06.moduleActive )
   END_RUNG wire#w7
   RUNG wire#w7
      I_Contact( "EM01".PackML_Sts.CM07.moduleActive )
   END_RUNG wire#w8
   RUNG wire#w8
      I_Contact( "EM01".PackML_Sts.CM08.moduleActive )
   END_RUNG wire#w9
   RUNG wire#w9
      I_Contact( "EM01".PackML_Sts.CM09.moduleActive )
   END_RUNG wire#w10
   RUNG wire#w10
      I_Contact( "EM01".PackML_Sts.CM10.moduleActive )
   END_RUNG wire#w11
   // the same network as SCL:
   "EM01".PackML_Sts.Unit.sts_UnSuspending_SC := ("EM01".PackML_Sts.Alarm.sts_UnSuspending_SC OR NOT "EM01".PackML_Sts.Alarm.moduleActive) AND ("EM01".PackML_Sts.CM01.sts_UnSuspending_SC OR NOT "EM01".PackML_Sts.CM01.moduleActive) AND ("EM01".PackML_Sts.CM02.sts_UnSuspending_SC OR NOT "EM01".PackML_Sts.CM02.moduleActive) AND ("EM01".PackML_Sts.CM03.sts_UnSuspending_SC OR NOT "EM01".PackML_Sts.CM03.moduleActive) AND ("EM01".PackML_Sts.CM04.sts_UnSuspending_SC OR NOT "EM01".PackML_Sts.CM04.moduleActive) AND ("EM01".PackML_Sts.CM05.sts_UnSuspending_SC OR NOT "EM01".PackML_Sts.CM05.moduleActive) AND ("EM01".PackML_Sts.CM06.sts_UnSuspending_SC OR NOT "EM01".PackML_Sts.CM06.moduleActive) AND ("EM01".PackML_Sts.CM07.sts_UnSuspending_SC OR NOT "EM01".PackML_Sts.CM07.moduleActive) AND ("EM01".PackML_Sts.CM08.sts_UnSuspending_SC OR NOT "EM01".PackML_Sts.CM08.moduleActive) AND ("EM01".PackML_Sts.CM09.sts_UnSuspending_SC OR NOT "EM01".PackML_Sts.CM09.moduleActive) AND ("EM01".PackML_Sts.CM10.sts_UnSuspending_SC OR NOT "EM01".PackML_Sts.CM10.moduleActive);
END_REGION

REGION Network 15: EM - Abort Command
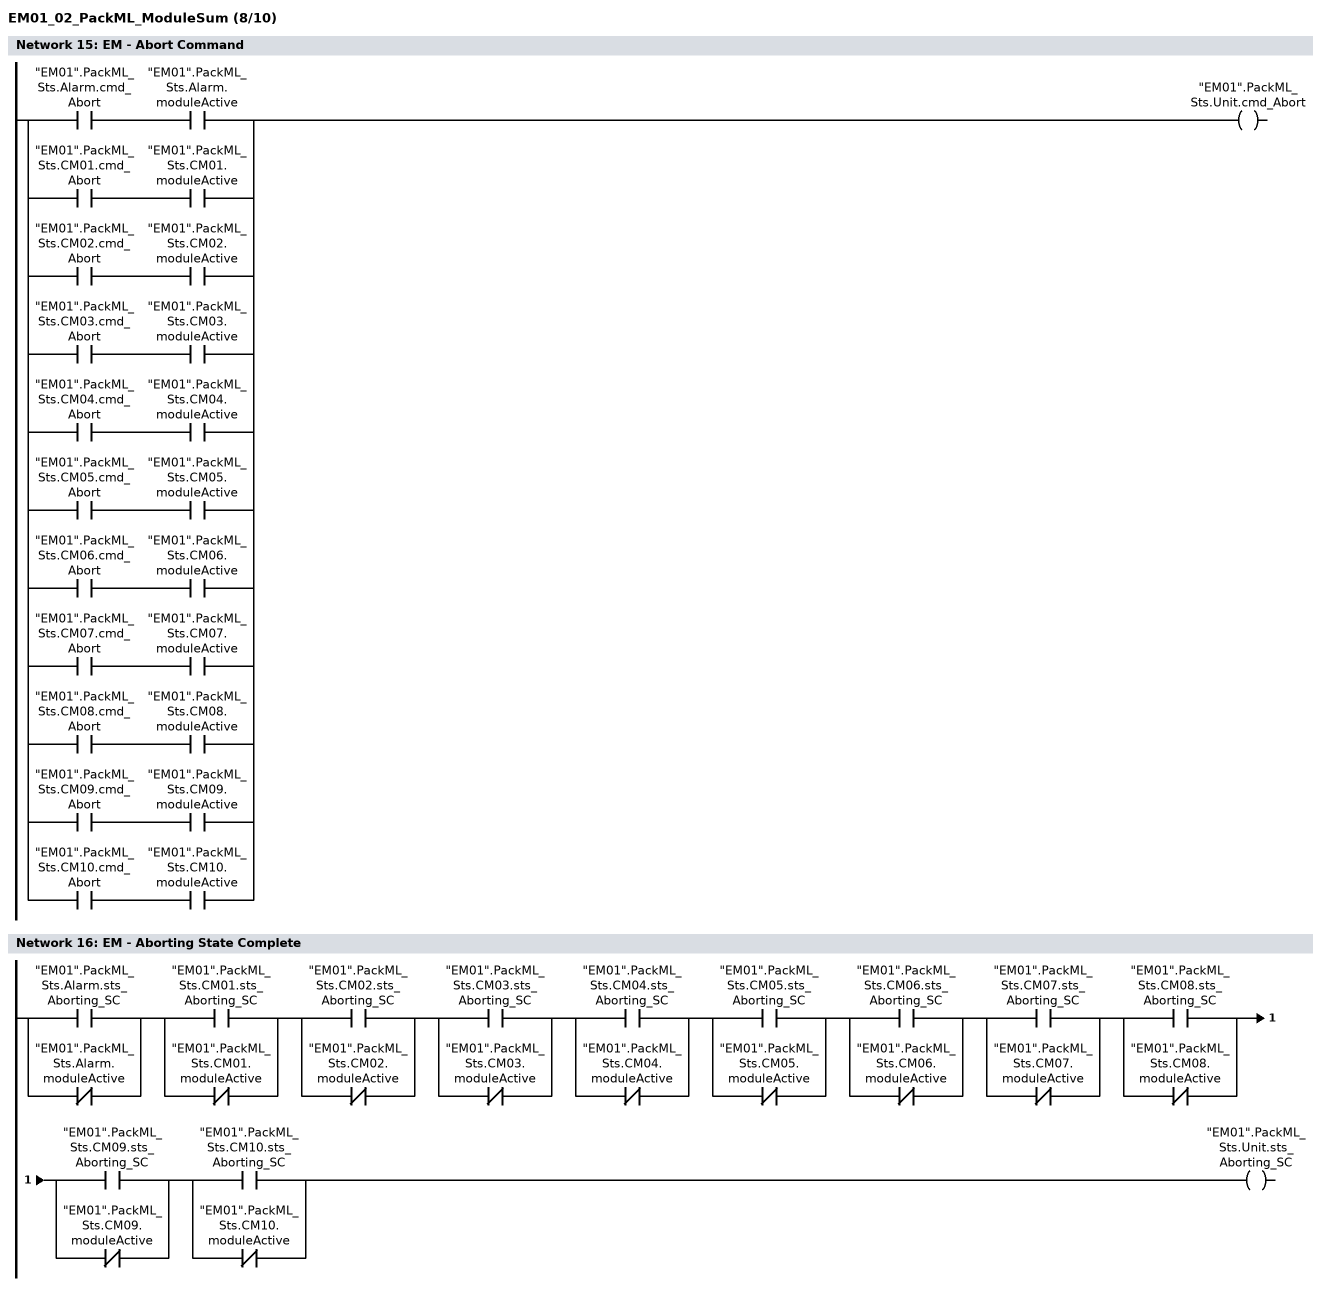
   RUNG wire#powerrail
      Contact( "EM01".PackML_Sts.Alarm.cmd_Abort )
      Contact( "EM01".PackML_Sts.Alarm.moduleActive )
      wire#w1
      Coil( "EM01".PackML_Sts.Unit.cmd_Abort )
   END_RUNG
   RUNG wire#powerrail
      Contact( "EM01".PackML_Sts.CM01.cmd_Abort )
      Contact( "EM01".PackML_Sts.CM01.moduleActive )
   END_RUNG wire#w1
   RUNG wire#powerrail
      Contact( "EM01".PackML_Sts.CM02.cmd_Abort )
      Contact( "EM01".PackML_Sts.CM02.moduleActive )
   END_RUNG wire#w1
   RUNG wire#powerrail
      Contact( "EM01".PackML_Sts.CM03.cmd_Abort )
      Contact( "EM01".PackML_Sts.CM03.moduleActive )
   END_RUNG wire#w1
   RUNG wire#powerrail
      Contact( "EM01".PackML_Sts.CM04.cmd_Abort )
      Contact( "EM01".PackML_Sts.CM04.moduleActive )
   END_RUNG wire#w1
   RUNG wire#powerrail
      Contact( "EM01".PackML_Sts.CM05.cmd_Abort )
      Contact( "EM01".PackML_Sts.CM05.moduleActive )
   END_RUNG wire#w1
   RUNG wire#powerrail
      Contact( "EM01".PackML_Sts.CM06.cmd_Abort )
      Contact( "EM01".PackML_Sts.CM06.moduleActive )
   END_RUNG wire#w1
   RUNG wire#powerrail
      Contact( "EM01".PackML_Sts.CM07.cmd_Abort )
      Contact( "EM01".PackML_Sts.CM07.moduleActive )
   END_RUNG wire#w1
   RUNG wire#powerrail
      Contact( "EM01".PackML_Sts.CM08.cmd_Abort )
      Contact( "EM01".PackML_Sts.CM08.moduleActive )
   END_RUNG wire#w1
   RUNG wire#powerrail
      Contact( "EM01".PackML_Sts.CM09.cmd_Abort )
      Contact( "EM01".PackML_Sts.CM09.moduleActive )
   END_RUNG wire#w1
   RUNG wire#powerrail
      Contact( "EM01".PackML_Sts.CM10.cmd_Abort )
      Contact( "EM01".PackML_Sts.CM10.moduleActive )
   END_RUNG wire#w1
   // the same network as SCL:
   "EM01".PackML_Sts.Unit.cmd_Abort := ("EM01".PackML_Sts.Alarm.cmd_Abort AND "EM01".PackML_Sts.Alarm.moduleActive) OR ("EM01".PackML_Sts.CM01.cmd_Abort AND "EM01".PackML_Sts.CM01.moduleActive) OR ("EM01".PackML_Sts.CM02.cmd_Abort AND "EM01".PackML_Sts.CM02.moduleActive) OR ("EM01".PackML_Sts.CM03.cmd_Abort AND "EM01".PackML_Sts.CM03.moduleActive) OR ("EM01".PackML_Sts.CM04.cmd_Abort AND "EM01".PackML_Sts.CM04.moduleActive) OR ("EM01".PackML_Sts.CM05.cmd_Abort AND "EM01".PackML_Sts.CM05.moduleActive) OR ("EM01".PackML_Sts.CM06.cmd_Abort AND "EM01".PackML_Sts.CM06.moduleActive) OR ("EM01".PackML_Sts.CM07.cmd_Abort AND "EM01".PackML_Sts.CM07.moduleActive) OR ("EM01".PackML_Sts.CM08.cmd_Abort AND "EM01".PackML_Sts.CM08.moduleActive) OR ("EM01".PackML_Sts.CM09.cmd_Abort AND "EM01".PackML_Sts.CM09.moduleActive) OR ("EM01".PackML_Sts.CM10.cmd_Abort AND "EM01".PackML_Sts.CM10.moduleActive);
END_REGION

REGION Network 16: EM - Aborting State Complete
   RUNG wire#powerrail
      Contact( "EM01".PackML_Sts.Alarm.sts_Aborting_SC )
      wire#w1
      Contact( "EM01".PackML_Sts.CM01.sts_Aborting_SC )
      wire#w2
      Contact( "EM01".PackML_Sts.CM02.sts_Aborting_SC )
      wire#w3
      Contact( "EM01".PackML_Sts.CM03.sts_Aborting_SC )
      wire#w4
      Contact( "EM01".PackML_Sts.CM04.sts_Aborting_SC )
      wire#w5
      Contact( "EM01".PackML_Sts.CM05.sts_Aborting_SC )
      wire#w6
      Contact( "EM01".PackML_Sts.CM06.sts_Aborting_SC )
      wire#w7
      Contact( "EM01".PackML_Sts.CM07.sts_Aborting_SC )
      wire#w8
      Contact( "EM01".PackML_Sts.CM08.sts_Aborting_SC )
      wire#w9
      Contact( "EM01".PackML_Sts.CM09.sts_Aborting_SC )
      wire#w10
      Contact( "EM01".PackML_Sts.CM10.sts_Aborting_SC )
      wire#w11
      Coil( "EM01".PackML_Sts.Unit.sts_Aborting_SC )
   END_RUNG
   RUNG wire#powerrail
      I_Contact( "EM01".PackML_Sts.Alarm.moduleActive )
   END_RUNG wire#w1
   RUNG wire#w1
      I_Contact( "EM01".PackML_Sts.CM01.moduleActive )
   END_RUNG wire#w2
   RUNG wire#w2
      I_Contact( "EM01".PackML_Sts.CM02.moduleActive )
   END_RUNG wire#w3
   RUNG wire#w3
      I_Contact( "EM01".PackML_Sts.CM03.moduleActive )
   END_RUNG wire#w4
   RUNG wire#w4
      I_Contact( "EM01".PackML_Sts.CM04.moduleActive )
   END_RUNG wire#w5
   RUNG wire#w5
      I_Contact( "EM01".PackML_Sts.CM05.moduleActive )
   END_RUNG wire#w6
   RUNG wire#w6
      I_Contact( "EM01".PackML_Sts.CM06.moduleActive )
   END_RUNG wire#w7
   RUNG wire#w7
      I_Contact( "EM01".PackML_Sts.CM07.moduleActive )
   END_RUNG wire#w8
   RUNG wire#w8
      I_Contact( "EM01".PackML_Sts.CM08.moduleActive )
   END_RUNG wire#w9
   RUNG wire#w9
      I_Contact( "EM01".PackML_Sts.CM09.moduleActive )
   END_RUNG wire#w10
   RUNG wire#w10
      I_Contact( "EM01".PackML_Sts.CM10.moduleActive )
   END_RUNG wire#w11
   // the same network as SCL:
   "EM01".PackML_Sts.Unit.sts_Aborting_SC := ("EM01".PackML_Sts.Alarm.sts_Aborting_SC OR NOT "EM01".PackML_Sts.Alarm.moduleActive) AND ("EM01".PackML_Sts.CM01.sts_Aborting_SC OR NOT "EM01".PackML_Sts.CM01.moduleActive) AND ("EM01".PackML_Sts.CM02.sts_Aborting_SC OR NOT "EM01".PackML_Sts.CM02.moduleActive) AND ("EM01".PackML_Sts.CM03.sts_Aborting_SC OR NOT "EM01".PackML_Sts.CM03.moduleActive) AND ("EM01".PackML_Sts.CM04.sts_Aborting_SC OR NOT "EM01".PackML_Sts.CM04.moduleActive) AND ("EM01".PackML_Sts.CM05.sts_Aborting_SC OR NOT "EM01".PackML_Sts.CM05.moduleActive) AND ("EM01".PackML_Sts.CM06.sts_Aborting_SC OR NOT "EM01".PackML_Sts.CM06.moduleActive) AND ("EM01".PackML_Sts.CM07.sts_Aborting_SC OR NOT "EM01".PackML_Sts.CM07.moduleActive) AND ("EM01".PackML_Sts.CM08.sts_Aborting_SC OR NOT "EM01".PackML_Sts.CM08.moduleActive) AND ("EM01".PackML_Sts.CM09.sts_Aborting_SC OR NOT "EM01".PackML_Sts.CM09.moduleActive) AND ("EM01".PackML_Sts.CM10.sts_Aborting_SC OR NOT "EM01".PackML_Sts.CM10.moduleActive);
END_REGION

REGION Network 17: EM - Clear Command
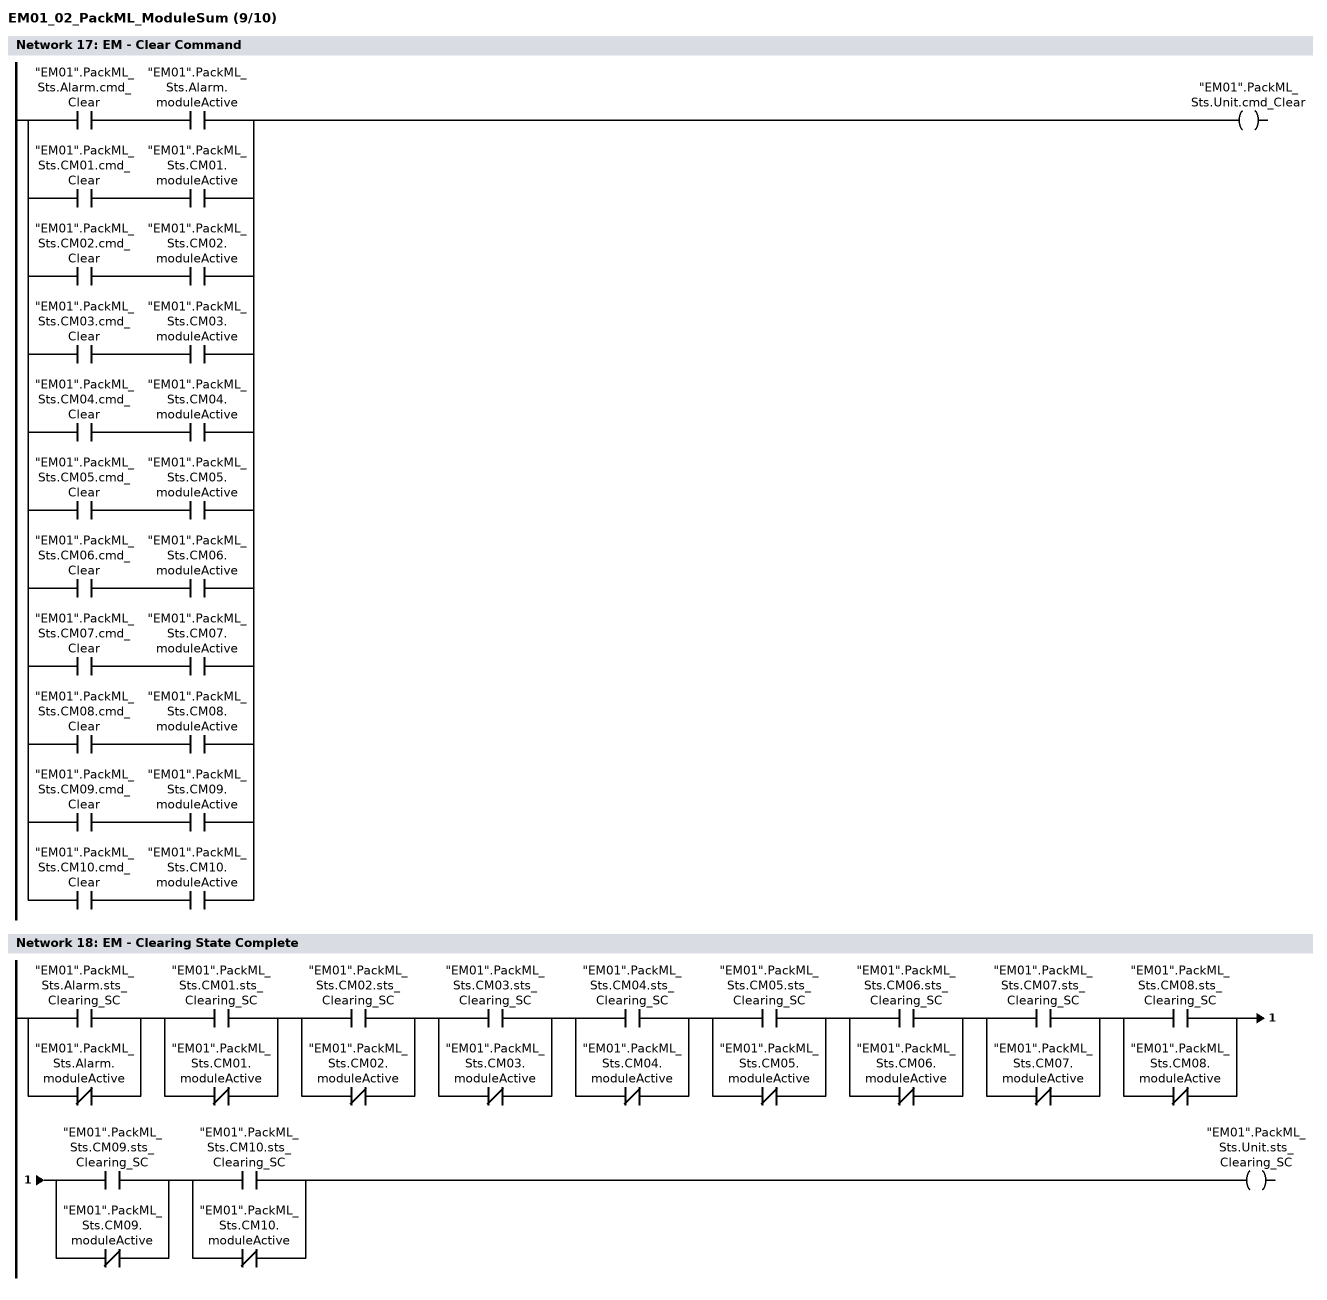
   RUNG wire#powerrail
      Contact( "EM01".PackML_Sts.Alarm.cmd_Clear )
      Contact( "EM01".PackML_Sts.Alarm.moduleActive )
      wire#w1
      Coil( "EM01".PackML_Sts.Unit.cmd_Clear )
   END_RUNG
   RUNG wire#powerrail
      Contact( "EM01".PackML_Sts.CM01.cmd_Clear )
      Contact( "EM01".PackML_Sts.CM01.moduleActive )
   END_RUNG wire#w1
   RUNG wire#powerrail
      Contact( "EM01".PackML_Sts.CM02.cmd_Clear )
      Contact( "EM01".PackML_Sts.CM02.moduleActive )
   END_RUNG wire#w1
   RUNG wire#powerrail
      Contact( "EM01".PackML_Sts.CM03.cmd_Clear )
      Contact( "EM01".PackML_Sts.CM03.moduleActive )
   END_RUNG wire#w1
   RUNG wire#powerrail
      Contact( "EM01".PackML_Sts.CM04.cmd_Clear )
      Contact( "EM01".PackML_Sts.CM04.moduleActive )
   END_RUNG wire#w1
   RUNG wire#powerrail
      Contact( "EM01".PackML_Sts.CM05.cmd_Clear )
      Contact( "EM01".PackML_Sts.CM05.moduleActive )
   END_RUNG wire#w1
   RUNG wire#powerrail
      Contact( "EM01".PackML_Sts.CM06.cmd_Clear )
      Contact( "EM01".PackML_Sts.CM06.moduleActive )
   END_RUNG wire#w1
   RUNG wire#powerrail
      Contact( "EM01".PackML_Sts.CM07.cmd_Clear )
      Contact( "EM01".PackML_Sts.CM07.moduleActive )
   END_RUNG wire#w1
   RUNG wire#powerrail
      Contact( "EM01".PackML_Sts.CM08.cmd_Clear )
      Contact( "EM01".PackML_Sts.CM08.moduleActive )
   END_RUNG wire#w1
   RUNG wire#powerrail
      Contact( "EM01".PackML_Sts.CM09.cmd_Clear )
      Contact( "EM01".PackML_Sts.CM09.moduleActive )
   END_RUNG wire#w1
   RUNG wire#powerrail
      Contact( "EM01".PackML_Sts.CM10.cmd_Clear )
      Contact( "EM01".PackML_Sts.CM10.moduleActive )
   END_RUNG wire#w1
   // the same network as SCL:
   "EM01".PackML_Sts.Unit.cmd_Clear := ("EM01".PackML_Sts.Alarm.cmd_Clear AND "EM01".PackML_Sts.Alarm.moduleActive) OR ("EM01".PackML_Sts.CM01.cmd_Clear AND "EM01".PackML_Sts.CM01.moduleActive) OR ("EM01".PackML_Sts.CM02.cmd_Clear AND "EM01".PackML_Sts.CM02.moduleActive) OR ("EM01".PackML_Sts.CM03.cmd_Clear AND "EM01".PackML_Sts.CM03.moduleActive) OR ("EM01".PackML_Sts.CM04.cmd_Clear AND "EM01".PackML_Sts.CM04.moduleActive) OR ("EM01".PackML_Sts.CM05.cmd_Clear AND "EM01".PackML_Sts.CM05.moduleActive) OR ("EM01".PackML_Sts.CM06.cmd_Clear AND "EM01".PackML_Sts.CM06.moduleActive) OR ("EM01".PackML_Sts.CM07.cmd_Clear AND "EM01".PackML_Sts.CM07.moduleActive) OR ("EM01".PackML_Sts.CM08.cmd_Clear AND "EM01".PackML_Sts.CM08.moduleActive) OR ("EM01".PackML_Sts.CM09.cmd_Clear AND "EM01".PackML_Sts.CM09.moduleActive) OR ("EM01".PackML_Sts.CM10.cmd_Clear AND "EM01".PackML_Sts.CM10.moduleActive);
END_REGION

REGION Network 18: EM - Clearing State Complete
   RUNG wire#powerrail
      Contact( "EM01".PackML_Sts.Alarm.sts_Clearing_SC )
      wire#w1
      Contact( "EM01".PackML_Sts.CM01.sts_Clearing_SC )
      wire#w2
      Contact( "EM01".PackML_Sts.CM02.sts_Clearing_SC )
      wire#w3
      Contact( "EM01".PackML_Sts.CM03.sts_Clearing_SC )
      wire#w4
      Contact( "EM01".PackML_Sts.CM04.sts_Clearing_SC )
      wire#w5
      Contact( "EM01".PackML_Sts.CM05.sts_Clearing_SC )
      wire#w6
      Contact( "EM01".PackML_Sts.CM06.sts_Clearing_SC )
      wire#w7
      Contact( "EM01".PackML_Sts.CM07.sts_Clearing_SC )
      wire#w8
      Contact( "EM01".PackML_Sts.CM08.sts_Clearing_SC )
      wire#w9
      Contact( "EM01".PackML_Sts.CM09.sts_Clearing_SC )
      wire#w10
      Contact( "EM01".PackML_Sts.CM10.sts_Clearing_SC )
      wire#w11
      Coil( "EM01".PackML_Sts.Unit.sts_Clearing_SC )
   END_RUNG
   RUNG wire#powerrail
      I_Contact( "EM01".PackML_Sts.Alarm.moduleActive )
   END_RUNG wire#w1
   RUNG wire#w1
      I_Contact( "EM01".PackML_Sts.CM01.moduleActive )
   END_RUNG wire#w2
   RUNG wire#w2
      I_Contact( "EM01".PackML_Sts.CM02.moduleActive )
   END_RUNG wire#w3
   RUNG wire#w3
      I_Contact( "EM01".PackML_Sts.CM03.moduleActive )
   END_RUNG wire#w4
   RUNG wire#w4
      I_Contact( "EM01".PackML_Sts.CM04.moduleActive )
   END_RUNG wire#w5
   RUNG wire#w5
      I_Contact( "EM01".PackML_Sts.CM05.moduleActive )
   END_RUNG wire#w6
   RUNG wire#w6
      I_Contact( "EM01".PackML_Sts.CM06.moduleActive )
   END_RUNG wire#w7
   RUNG wire#w7
      I_Contact( "EM01".PackML_Sts.CM07.moduleActive )
   END_RUNG wire#w8
   RUNG wire#w8
      I_Contact( "EM01".PackML_Sts.CM08.moduleActive )
   END_RUNG wire#w9
   RUNG wire#w9
      I_Contact( "EM01".PackML_Sts.CM09.moduleActive )
   END_RUNG wire#w10
   RUNG wire#w10
      I_Contact( "EM01".PackML_Sts.CM10.moduleActive )
   END_RUNG wire#w11
   // the same network as SCL:
   "EM01".PackML_Sts.Unit.sts_Clearing_SC := ("EM01".PackML_Sts.Alarm.sts_Clearing_SC OR NOT "EM01".PackML_Sts.Alarm.moduleActive) AND ("EM01".PackML_Sts.CM01.sts_Clearing_SC OR NOT "EM01".PackML_Sts.CM01.moduleActive) AND ("EM01".PackML_Sts.CM02.sts_Clearing_SC OR NOT "EM01".PackML_Sts.CM02.moduleActive) AND ("EM01".PackML_Sts.CM03.sts_Clearing_SC OR NOT "EM01".PackML_Sts.CM03.moduleActive) AND ("EM01".PackML_Sts.CM04.sts_Clearing_SC OR NOT "EM01".PackML_Sts.CM04.moduleActive) AND ("EM01".PackML_Sts.CM05.sts_Clearing_SC OR NOT "EM01".PackML_Sts.CM05.moduleActive) AND ("EM01".PackML_Sts.CM06.sts_Clearing_SC OR NOT "EM01".PackML_Sts.CM06.moduleActive) AND ("EM01".PackML_Sts.CM07.sts_Clearing_SC OR NOT "EM01".PackML_Sts.CM07.moduleActive) AND ("EM01".PackML_Sts.CM08.sts_Clearing_SC OR NOT "EM01".PackML_Sts.CM08.moduleActive) AND ("EM01".PackML_Sts.CM09.sts_Clearing_SC OR NOT "EM01".PackML_Sts.CM09.moduleActive) AND ("EM01".PackML_Sts.CM10.sts_Clearing_SC OR NOT "EM01".PackML_Sts.CM10.moduleActive);
END_REGION

REGION Network 19: EM - Execute State Complete
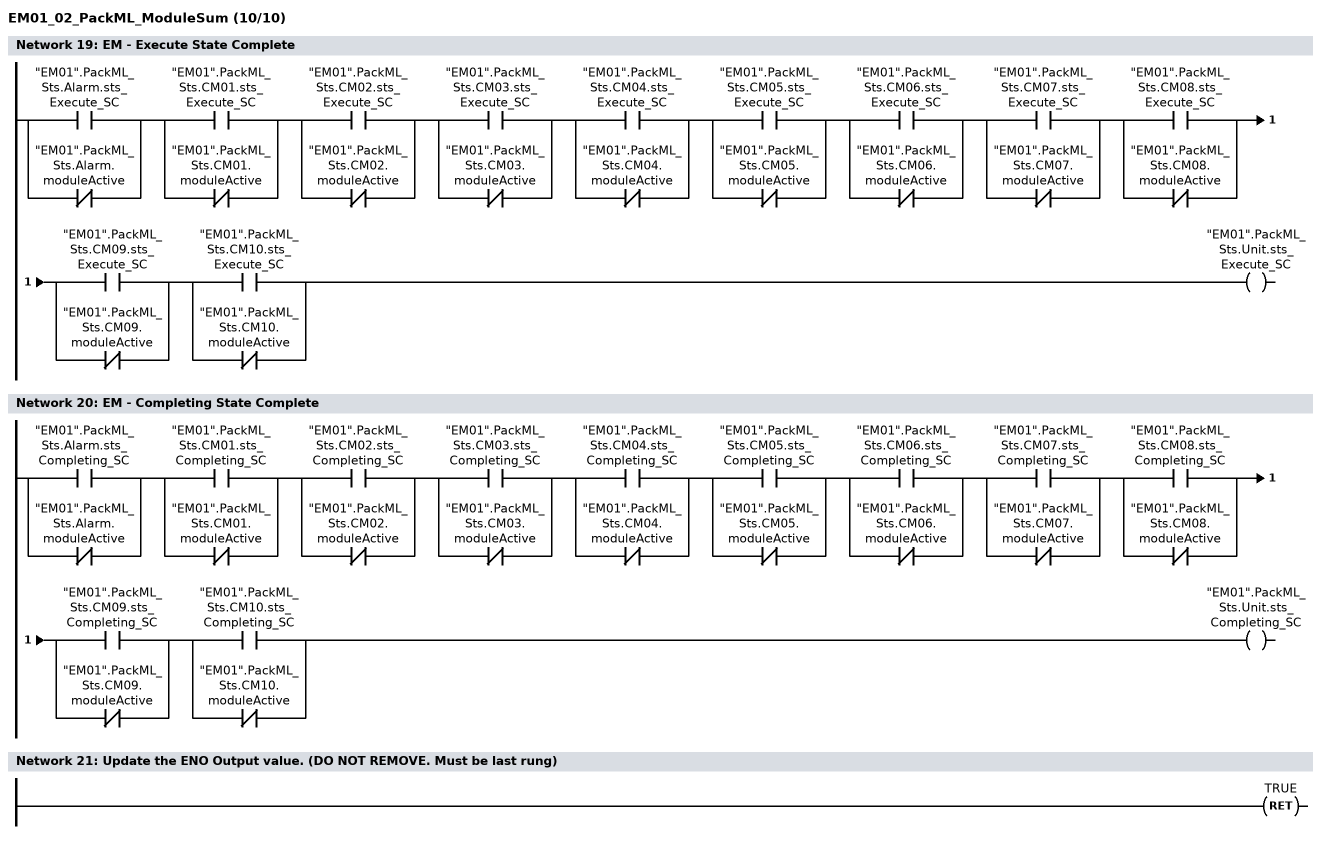
   RUNG wire#powerrail
      Contact( "EM01".PackML_Sts.Alarm.sts_Execute_SC )
      wire#w1
      Contact( "EM01".PackML_Sts.CM01.sts_Execute_SC )
      wire#w2
      Contact( "EM01".PackML_Sts.CM02.sts_Execute_SC )
      wire#w3
      Contact( "EM01".PackML_Sts.CM03.sts_Execute_SC )
      wire#w4
      Contact( "EM01".PackML_Sts.CM04.sts_Execute_SC )
      wire#w5
      Contact( "EM01".PackML_Sts.CM05.sts_Execute_SC )
      wire#w6
      Contact( "EM01".PackML_Sts.CM06.sts_Execute_SC )
      wire#w7
      Contact( "EM01".PackML_Sts.CM07.sts_Execute_SC )
      wire#w8
      Contact( "EM01".PackML_Sts.CM08.sts_Execute_SC )
      wire#w9
      Contact( "EM01".PackML_Sts.CM09.sts_Execute_SC )
      wire#w10
      Contact( "EM01".PackML_Sts.CM10.sts_Execute_SC )
      wire#w11
      Coil( "EM01".PackML_Sts.Unit.sts_Execute_SC )
   END_RUNG
   RUNG wire#powerrail
      I_Contact( "EM01".PackML_Sts.Alarm.moduleActive )
   END_RUNG wire#w1
   RUNG wire#w1
      I_Contact( "EM01".PackML_Sts.CM01.moduleActive )
   END_RUNG wire#w2
   RUNG wire#w2
      I_Contact( "EM01".PackML_Sts.CM02.moduleActive )
   END_RUNG wire#w3
   RUNG wire#w3
      I_Contact( "EM01".PackML_Sts.CM03.moduleActive )
   END_RUNG wire#w4
   RUNG wire#w4
      I_Contact( "EM01".PackML_Sts.CM04.moduleActive )
   END_RUNG wire#w5
   RUNG wire#w5
      I_Contact( "EM01".PackML_Sts.CM05.moduleActive )
   END_RUNG wire#w6
   RUNG wire#w6
      I_Contact( "EM01".PackML_Sts.CM06.moduleActive )
   END_RUNG wire#w7
   RUNG wire#w7
      I_Contact( "EM01".PackML_Sts.CM07.moduleActive )
   END_RUNG wire#w8
   RUNG wire#w8
      I_Contact( "EM01".PackML_Sts.CM08.moduleActive )
   END_RUNG wire#w9
   RUNG wire#w9
      I_Contact( "EM01".PackML_Sts.CM09.moduleActive )
   END_RUNG wire#w10
   RUNG wire#w10
      I_Contact( "EM01".PackML_Sts.CM10.moduleActive )
   END_RUNG wire#w11
   // the same network as SCL:
   "EM01".PackML_Sts.Unit.sts_Execute_SC := ("EM01".PackML_Sts.Alarm.sts_Execute_SC OR NOT "EM01".PackML_Sts.Alarm.moduleActive) AND ("EM01".PackML_Sts.CM01.sts_Execute_SC OR NOT "EM01".PackML_Sts.CM01.moduleActive) AND ("EM01".PackML_Sts.CM02.sts_Execute_SC OR NOT "EM01".PackML_Sts.CM02.moduleActive) AND ("EM01".PackML_Sts.CM03.sts_Execute_SC OR NOT "EM01".PackML_Sts.CM03.moduleActive) AND ("EM01".PackML_Sts.CM04.sts_Execute_SC OR NOT "EM01".PackML_Sts.CM04.moduleActive) AND ("EM01".PackML_Sts.CM05.sts_Execute_SC OR NOT "EM01".PackML_Sts.CM05.moduleActive) AND ("EM01".PackML_Sts.CM06.sts_Execute_SC OR NOT "EM01".PackML_Sts.CM06.moduleActive) AND ("EM01".PackML_Sts.CM07.sts_Execute_SC OR NOT "EM01".PackML_Sts.CM07.moduleActive) AND ("EM01".PackML_Sts.CM08.sts_Execute_SC OR NOT "EM01".PackML_Sts.CM08.moduleActive) AND ("EM01".PackML_Sts.CM09.sts_Execute_SC OR NOT "EM01".PackML_Sts.CM09.moduleActive) AND ("EM01".PackML_Sts.CM10.sts_Execute_SC OR NOT "EM01".PackML_Sts.CM10.moduleActive);
END_REGION

REGION Network 20: EM - Completing State Complete
   RUNG wire#powerrail
      Contact( "EM01".PackML_Sts.Alarm.sts_Completing_SC )
      wire#w1
      Contact( "EM01".PackML_Sts.CM01.sts_Completing_SC )
      wire#w2
      Contact( "EM01".PackML_Sts.CM02.sts_Completing_SC )
      wire#w3
      Contact( "EM01".PackML_Sts.CM03.sts_Completing_SC )
      wire#w4
      Contact( "EM01".PackML_Sts.CM04.sts_Completing_SC )
      wire#w5
      Contact( "EM01".PackML_Sts.CM05.sts_Completing_SC )
      wire#w6
      Contact( "EM01".PackML_Sts.CM06.sts_Completing_SC )
      wire#w7
      Contact( "EM01".PackML_Sts.CM07.sts_Completing_SC )
      wire#w8
      Contact( "EM01".PackML_Sts.CM08.sts_Completing_SC )
      wire#w9
      Contact( "EM01".PackML_Sts.CM09.sts_Completing_SC )
      wire#w10
      Contact( "EM01".PackML_Sts.CM10.sts_Completing_SC )
      wire#w11
      Coil( "EM01".PackML_Sts.Unit.sts_Completing_SC )
   END_RUNG
   RUNG wire#powerrail
      I_Contact( "EM01".PackML_Sts.Alarm.moduleActive )
   END_RUNG wire#w1
   RUNG wire#w1
      I_Contact( "EM01".PackML_Sts.CM01.moduleActive )
   END_RUNG wire#w2
   RUNG wire#w2
      I_Contact( "EM01".PackML_Sts.CM02.moduleActive )
   END_RUNG wire#w3
   RUNG wire#w3
      I_Contact( "EM01".PackML_Sts.CM03.moduleActive )
   END_RUNG wire#w4
   RUNG wire#w4
      I_Contact( "EM01".PackML_Sts.CM04.moduleActive )
   END_RUNG wire#w5
   RUNG wire#w5
      I_Contact( "EM01".PackML_Sts.CM05.moduleActive )
   END_RUNG wire#w6
   RUNG wire#w6
      I_Contact( "EM01".PackML_Sts.CM06.moduleActive )
   END_RUNG wire#w7
   RUNG wire#w7
      I_Contact( "EM01".PackML_Sts.CM07.moduleActive )
   END_RUNG wire#w8
   RUNG wire#w8
      I_Contact( "EM01".PackML_Sts.CM08.moduleActive )
   END_RUNG wire#w9
   RUNG wire#w9
      I_Contact( "EM01".PackML_Sts.CM09.moduleActive )
   END_RUNG wire#w10
   RUNG wire#w10
      I_Contact( "EM01".PackML_Sts.CM10.moduleActive )
   END_RUNG wire#w11
   // the same network as SCL:
   "EM01".PackML_Sts.Unit.sts_Completing_SC := ("EM01".PackML_Sts.Alarm.sts_Completing_SC OR NOT "EM01".PackML_Sts.Alarm.moduleActive) AND ("EM01".PackML_Sts.CM01.sts_Completing_SC OR NOT "EM01".PackML_Sts.CM01.moduleActive) AND ("EM01".PackML_Sts.CM02.sts_Completing_SC OR NOT "EM01".PackML_Sts.CM02.moduleActive) AND ("EM01".PackML_Sts.CM03.sts_Completing_SC OR NOT "EM01".PackML_Sts.CM03.moduleActive) AND ("EM01".PackML_Sts.CM04.sts_Completing_SC OR NOT "EM01".PackML_Sts.CM04.moduleActive) AND ("EM01".PackML_Sts.CM05.sts_Completing_SC OR NOT "EM01".PackML_Sts.CM05.moduleActive) AND ("EM01".PackML_Sts.CM06.sts_Completing_SC OR NOT "EM01".PackML_Sts.CM06.moduleActive) AND ("EM01".PackML_Sts.CM07.sts_Completing_SC OR NOT "EM01".PackML_Sts.CM07.moduleActive) AND ("EM01".PackML_Sts.CM08.sts_Completing_SC OR NOT "EM01".PackML_Sts.CM08.moduleActive) AND ("EM01".PackML_Sts.CM09.sts_Completing_SC OR NOT "EM01".PackML_Sts.CM09.moduleActive) AND ("EM01".PackML_Sts.CM10.sts_Completing_SC OR NOT "EM01".PackML_Sts.CM10.moduleActive);
END_REGION

REGION Network 21: Update the ENO Output value. (DO NOT REMOVE. Must be last rung)
   RUNG wire#powerrail
      ReturnCoil( TRUE )
   END_RUNG
   // the same network as SCL:
   ENO := TRUE;
   RETURN;
END_REGION
END_FUNCTION_BLOCK
